(* IEC 61131-3 sources: std_i2980_v2.06_cp053/Source/IMM/ieccontrol/GlobalBaseArchives (part 9) *)

@END_Body

@@@BEG_Comment@@@
@TL(3)
This Algo receives the evCheckLocklist event,
checks the startconditions for the movement and outputs alarms if it is not allowed.
The movement itself is not started.
@@@END_Comment@@@

@BEG_Body
@TL(57)
(**************************************** WARNING ********************************************
 *** The KEBA Kemro K2 System including software is not intended for safety control tasks! ***
 ***                       For further information see Comment tab!                        ***
 *********************************************************************************************)

IF (evLockGroupEnableDisableData.DeviceIdReceiver.CompId = sv_DeviceId.CompId OR evLockGroupEnableDisableData.DeviceIdReceiver.CompId = cCompAll) AND
   (evLockGroupEnableDisableData.DeviceIdReceiver.IndexId = sv_DeviceId.IndexId OR evLockGroupEnableDisableData.DeviceIdReceiver.IndexId = cAllDevIndex) THEN

   //check all registered movements if the sent MoveDir and MoveId are equal
   FOR i := 1 TO sv_NumberOfMovements DO

      IF ((sv_Movements[i]^.MoveDir = evLockGroupEnableDisableData.MoveDir) OR (evLockGroupEnableDisableData.MoveDir = cMoveAll)) AND
         ((sv_Movements[i]^.MoveId = evLockGroupEnableDisableData.MoveId) OR (evLockGroupEnableDisableData.MoveId = cMoveAll)) THEN

         //check if this movement is a member of the sent lockgroup
         FOR j := 1 TO cMaxGroupLocks DO

            IF sv_Movements[i]^.LockGroups[j] = evLockGroupEnableDisableData.LockGroup THEN
               IF evLockGroupEnableDisableData.Mode = nLockGroupDisable THEN
                  mDisabledLockGroups[i][j] := TRUE;
               ELSE
                  mDisabledLockGroups[i][j] := FALSE;
               END_IF;

               IF sv_TraceLevel.bLockUnlock THEN
                  IF mDisabledLockGroups[i][j] THEN
                     sMode := ' disabled';
                  ELSE
                     sMode := ' enabled';
                  END_IF;

                  fbDebugTrace(CONCAT('lockgroup ', DINT_TO_STRING(evLockGroupEnableDisableData.LockGroup), ' of movement ',
                        DINT_TO_STRING(sv_Movements[i]^.MoveDir), '/', DINT_TO_STRING(sv_Movements[i]^.MoveId),
                        sMode, ' by Device ', DINT_TO_STRING(evLockGroupEnableDisableData.DeviceIdSender.CompId),
                        '.', DINT_TO_STRING(evLockGroupEnableDisableData.DeviceIdSender.IndexId)));
               END_IF;

               //update locklist
               abLockList.aUpdateLockDisable.Entry.DeviceIdSender := evLockGroupEnableDisableData.DeviceIdSender;
               abLockList.aUpdateLockDisable.Entry.MoveDir := sv_Movements[i]^.MoveDir;
               abLockList.aUpdateLockDisable.Entry.MoveId := sv_Movements[i]^.MoveId;
               abLockList.aUpdateLockDisable.Entry.Alarm := evLockGroupEnableDisableData.Alarm;
               abLockList.aUpdateLockDisable.bDisable := mDisabledLockGroups[i][j];
               abLockList.aUpdateLockDisable();
               EXIT;
            END_IF;

         END_FOR;  //end_for check lockgroups of the movement
      END_IF;  //end_if MoveDir and MoveId fit to event data
   END_FOR; //end_for check all movements

END_IF;

@END_Body

@@@BEG_Comment@@@
@TL(3)
receives evLockGroupEnableDisable event and updates locklist
if a registered movement of this function unit is a member of the
specified lockgroup
@@@END_Comment@@@
@END_Body

@END_Contents

(* ---- ABDeviceRegister.pu ---- *)
(*
@h    ! WARNING !
@h    The Kemro K2 system (including software) only meets category B according to EN 954-1,
@h    thus it is not intended for usage in safety-relevant control applications in the field
@h    of personal safety (e.g. emergency stop).
@h    To implement potentially necessary safety-relevant control tasks, always use additional
@h    external safety devices that are intended for the particular purpose, and meet the necessary
@h    functional safety.
@h    For further information see EN 954-1 (EN ISO 13849-1) and/or the K2-x00 user manual, chapter
@h    "CE conformity, directives and standards".

Increments the registration counter and calls the deviceregistation after the registrationdelay is up.
Every instance of ABDeviceRegister gets another delaytime - to give the other FUs time to increment
the registration counter.
*)

IMPORT_OVER_LISTFILE
 ABRegisterDelay
, FBDeviceRegister

END_IMPORT

ALGORITHM_BLOCK ABDeviceRegister #DUMMY_EDIT_BLOCK

SYSTEM_VAR
 sv_iDevicesToRegister : DINT;
END_VAR

SYSTEM_OBJECT
 Task10ms : TASK;
END_OBJECT

(*
Deviceregistration
*)

PROCESS_ALGORITHM paInit ON Task10ms AUTOSTART

VAR
 abRegisterDelay : ABRegisterDelay;
 fbDeviceRegister : FBDeviceRegister;
END_VAR

(* IecGraph-Code *)

(* init step *)
INITIAL_STEP DELAY:
aGetDelayTime (P);
END_STEP

ACTION aGetDelayTime: #BEGIN_EDIT_BLOCK
sv_iDevicesToRegister := sv_iDevicesToRegister + 1;
abRegisterDelay.aGet();

;#END_EDIT_BLOCK END_ACTION (*aGetDelayTime*)

(* steps *)
STEP DEVICE_REG:
Action2 (P);
END_STEP

ACTION Action2: #BEGIN_EDIT_BLOCK
fbDeviceRegister();
STOP_PROCESS_ALGORITHM();

;#END_EDIT_BLOCK END_ACTION (*Action2*)

(* transitions *)
TRANSITION Trans1 FROM DELAY TO DEVICE_REG :=  #BEGIN_EDIT_BLOCK
DELAY.T >= abRegisterDelay.aGet.Time
;#END_EDIT_BLOCK
END_TRANSITION

(* end IecGraph-Code *)
(* sfc-code *)
(* end sfc-code *)

END_ALGORITHM

END_ALGORITHM_BLOCK

#END_OF_IEC_PART

@Puma @IecEditor 6 10 @Pou 25
@@@BEG_Comment@@@
@h    ! WARNING !
@h    The Kemro K2 system (including software) only meets category B according to EN 954-1,
@h    thus it is not intended for usage in safety-relevant control applications in the field
@h    of personal safety (e.g. emergency stop).
@h    To implement potentially necessary safety-relevant control tasks, always use additional
@h    external safety devices that are intended for the particular purpose, and meet the necessary
@h    functional safety.
@h    For further information see EN 954-1 (EN ISO 13849-1) and/or the K2-x00 user manual, chapter
@h    "CE conformity, directives and standards".

Increments the registration counter and calls the deviceregistation after the registrationdelay is up.
Every instance of ABDeviceRegister gets another delaytime - to give the other FUs time to increment
the registration counter.
@@@END_Comment@@@

@BEG_Contents

@BEG_Func
@RT(17)FuncTreeContainer
0
@END_Func

@BEG_Const
@RT(18)ConstTreeContainer
0
@END_Const

@BEG_Export

@BEG_Kind
@ALGORITHM_BLOCK @RT(16)ABDeviceRegister @STRUCTURED_TEXT
@RT(0) @RT(0) @RT(0)
@END_Kind

@BEG_Dcl
@RT(16)DclTreeContainer
2
@Var @RT(21)sv_iDevicesToRegister @RT(0) @T @F @DT @RT(4)DINT @RT(0) @T @T @BASIC 0 @F
@F @F
@T
@BEG_Attrib
3 @RT(0) @RT(0) @RT(0)
@END_Attrib
1 8 @F @F @F @F

@Var @RT(8)Task10ms @RT(0) @T @T @RENAMED 0 @T @T @DT @RT(4)TASK @RT(0) @T @T @BASIC 0 @F
@F @F
@T
@BEG_Attrib
3 @RT(0) @RT(0) @RT(0)
@END_Attrib
1 7 @F @F @F @F

@END_Dcl

@END_Export

@BEG_Body

1

@BEG_Export

@BEG_Algo
@PROCESS_ALGORITHM @RT(6)paInit @SEQUENTIAL_FLOW_CHART
@RT(0) @RT(0) @RT(8)Task10ms @T @F
@END_Algo

@BEG_Dcl
@RT(16)DclTreeContainer
2
@Var @RT(15)abRegisterDelay @RT(0) @T @T @DERIVED 0 @T @T @DT @RT(15)ABRegisterDelay @RT(0) @T @T @UNKNOWN 0 @F
@F @F
@T
@BEG_Attrib
3 @RT(0) @RT(0) @RT(0)
@END_Attrib
1 0 @F @F @F @F

@Var @RT(16)fbDeviceRegister @RT(0) @T @T @DERIVED 0 @T @T @DT @RT(16)FBDeviceRegister @RT(0) @T @T @UNKNOWN 0 @F
@F @F
@T
@BEG_Attrib
3 @RT(0) @RT(0) @RT(0)
@END_Attrib
1 0 @F @F @F @F

@END_Dcl

@END_Export

@BEG_SfcBody
5 5 4

@BEG_SfcData 2
@StepSeq @RT(4)sseq @F 3
@Step @RT(5)DELAY @F @T @F @F @RT(0) @F
@AcbCont @RT(7)unnamed @F 1
@Acb @RT(13)aGetDelayTime @F @T @RT(1)P @RT(0) @F @F @T @TL(3)
sv_iDevicesToRegister := sv_iDevicesToRegister + 1;
abRegisterDelay.aGet();

@F

@Trans @RT(6)Trans1 @F @T @F @F @T @T @TL(2)
DELAY.T >= abRegisterDelay.aGet.Time

@RT(6)Trans1 @F
@Step @RT(10)DEVICE_REG @F @F @F @F @RT(0) @F
@AcbCont @RT(7)unnamed @F 1
@Acb @RT(7)Action2 @F @T @RT(1)P @RT(0) @F @F @T @TL(3)
fbDeviceRegister();
STOP_PROCESS_ALGORITHM();

@F

@END_SfcData
@SaActions 0
@SaTrans 0
@SaExits 0
@END_SfcBody

@@@BEG_Comment@@@
@TL(1)
Deviceregistration
@@@END_Comment@@@
@END_Body

@END_Contents

(* ---- ABEndPosMon.pu ---- *)
(*
@h    ! WARNING !
@h    The Kemro K2 system (including software) only meets category B according to EN 954-1,
@h    thus it is not intended for usage in safety-relevant control applications in the field
@h    of personal safety (e.g. emergency stop).
@h    To implement potentially necessary safety-relevant control tasks, always use additional
@h    external safety devices that are intended for the particular purpose, and meet the necessary
@h    functional safety.
@h    For further information see EN 954-1 (EN ISO 13849-1) and/or the K2-x00 user manual, chapter
@h    "CE conformity, directives and standards".

This AB is used for endposition supervision.
There are two possibilities to detect if an endpoint is reached.
- a limit switch for the endposition is available
- the last point of the entered movement profile is reached
The AB can handle a standard movement profile and plast profile.

The AB gives the following results in this cases:
1) only a limit switch and no movement profile
   => endposition is reached if limit switch is true

2) movement profile and no limit switch
   => endposition is reached if actual position is lower or equal / bigger or equal
      (depending on the movedirection) than last last position of the profile;
      a given tolerance will also be considered

3) movement profile and limit switch available
   => endposition is reached if both criterias from above are fullfilled
*)

IMPORT_OVER_LISTFILE
 CHECK_REF
, tsEndPosData
, KAPPL_VisProfile
, KAPPL_VisProfilePlast

END_IMPORT

ALGORITHM_BLOCK ABEndPosMon #DUMMY_EDIT_BLOCK

SYSTEM_VAR
 sv_EndPosData : tsEndPosData;
 sv_bInitStart : BOOL;
END_VAR

SYSTEM_OBJECT
 TaskAnalog : TASK;
 PU_Task_7 : TASK;
END_OBJECT

VAR
 mpProfile : REFTO KAPPL_VisProfile;
 mpPlastProfile : REFTO KAPPL_VisProfilePlast;
 mpTolerance : REFTO REAL;
 mbReparam : BOOL;
END_VAR

(*
This block checks if the actual position is within a tolerance at the target position.
If this condition is met, "Position Reached" is signaled.
*)

PROCESS_ALGORITHM paRun ON TaskAnalog(3000)

VAR
 bTargetPosReached : BOOL;
 rTargetPos : REAL;
 bDirection : BOOL;
 rTriggerPos : REAL;
 pbDI : REFTO BOOL;
 bDIConnected : BOOL;
 bValidMoveProfile : BOOL;
 bValidPlastProfile : BOOL;
 bValidProfile : BOOL;
 bInvertDI : BOOL;
END_VAR
#BEGIN_EDIT_BLOCK
(**************************************** WARNING ********************************************
 *** The KEBA Kemro K2 System including software is not intended for safety control tasks! ***
 ***                       For further information see Comment tab!                        ***
 *********************************************************************************************)

IF mbReparam THEN

   mpProfile := sv_EndPosData.pProfile;
   bValidMoveProfile := CHECK_REF(mpProfile^);
   mpPlastProfile := sv_EndPosData.pPlastProfile;
   bValidPlastProfile := CHECK_REF(mpPlastProfile^);
   bValidProfile := bValidMoveProfile OR bValidPlastProfile;

   pbDI := sv_EndPosData.pbDI;
   bDIConnected := CHECK_REF(pbDI^);
   bInvertDI := sv_EndPosData.bInvertDI;

   //get target position and direction
   IF bValidMoveProfile THEN
      rTargetPos := MAX(0.0, mpProfile^.Profile.Points[(mpProfile^.Profile.iNoOfPoints+1)].rStartPos);
      bDirection := mpProfile^.Profile.Points[mpProfile^.Profile.iNoOfPoints+1].rStartPos > mpProfile^.Profile.Points[1].rStartPos;
   ELSIF bValidPlastProfile THEN
      rTargetPos := MAX(0.0, mpPlastProfile^.Profile.Points[(mpPlastProfile^.Profile.iNoOfPoints+1)].rStartPos);
      bDirection := TRUE;
   END_IF;

   IF bValidProfile THEN
      IF bDirection THEN
         rTriggerPos := rTargetPos - sv_EndPosData.rTolerance^;
      ELSE
         rTriggerPos := rTargetPos + sv_EndPosData.rTolerance^;
      END_IF;
   END_IF;

   mbReparam := FALSE;
END_IF;

//cyclic part
IF bValidProfile THEN
   IF bDirection THEN
      bTargetPosReached := (sv_EndPosData.rActPos^ > rTriggerPos);
   ELSE
      bTargetPosReached := (sv_EndPosData.rActPos^ < rTriggerPos);
   END_IF;
END_IF;

IF bValidProfile AND bDIConnected THEN
   // profile and DI connected
   sv_EndPosData.pbPosReached^ := bTargetPosReached AND (pbDI^ XOR bInvertDI);
ELSIF bValidProfile THEN
   //only profile connected
   sv_EndPosData.pbPosReached^ := bTargetPosReached;
ELSIF bDIConnected THEN
   //only DI connected
   sv_EndPosData.pbPosReached^ := pbDI^ XOR bInvertDI;
END_IF;

;#END_EDIT_BLOCK END_ALGORITHM

POSTUPDATE_ALGORITHM pParameterChanged ON PU_Task_7 WITH mpTolerance^,mpProfile^.Profile,mpPlastProfile^.Profile,sv_EndPosData.pProfile,sv_EndPosData.pPlastProfile,sv_EndPosData.pbDI,sv_EndPosData.bInvertDI

#BEGIN_EDIT_BLOCK
(**************************************** WARNING ********************************************
 *** The KEBA Kemro K2 System including software is not intended for safety control tasks! ***
 ***                       For further information see Comment tab!                        ***
 *********************************************************************************************)

mbReparam := TRUE;

;#END_EDIT_BLOCK END_ALGORITHM

POSTUPDATE_ALGORITHM pInit ON PU_Task_7 WITH sv_bInitStart

#BEGIN_EDIT_BLOCK
(**************************************** WARNING ********************************************
 *** The KEBA Kemro K2 System including software is not intended for safety control tasks! ***
 ***                       For further information see Comment tab!                        ***
 *********************************************************************************************)

mpTolerance := sv_EndPosData.rTolerance;
mbReparam := TRUE;

START_PROCESS_ALGORITHM(paRun);

;#END_EDIT_BLOCK END_ALGORITHM

END_ALGORITHM_BLOCK

#END_OF_IEC_PART

@Puma @IecEditor 6 97 @Pou 25
@@@BEG_Comment@@@
@h    ! WARNING !
@h    The Kemro K2 system (including software) only meets category B according to EN 954-1,
@h    thus it is not intended for usage in safety-relevant control applications in the field
@h    of personal safety (e.g. emergency stop).
@h    To implement potentially necessary safety-relevant control tasks, always use additional
@h    external safety devices that are intended for the particular purpose, and meet the necessary
@h    functional safety.
@h    For further information see EN 954-1 (EN ISO 13849-1) and/or the K2-x00 user manual, chapter
@h    "CE conformity, directives and standards".

This AB is used for endposition supervision.
There are two possibilities to detect if an endpoint is reached.
- a limit switch for the endposition is available
- the last point of the entered movement profile is reached
The AB can handle a standard movement profile and plast profile.

The AB gives the following results in this cases:
1) only a limit switch and no movement profile
   => endposition is reached if limit switch is true

2) movement profile and no limit switch
   => endposition is reached if actual position is lower or equal / bigger or equal
      (depending on the movedirection) than last last position of the profile;
      a given tolerance will also be considered

3) movement profile and limit switch available
   => endposition is reached if both criterias from above are fullfilled
@@@END_Comment@@@

@BEG_Contents

@BEG_Func
@RT(17)FuncTreeContainer
1
@Var @RT(9)CHECK_REF @RT(0) @T @T @DERIVED 0 @F @RT(23)KEBA_STANDARD_PROCEDURE @F
@T
@BEG_Attrib
0 @RT(0) @RT(0)
@END_Attrib
1 1 @F @F @F @F

@END_Func

@BEG_Const
@RT(18)ConstTreeContainer
0
@END_Const

@BEG_Export

@BEG_Kind
@ALGORITHM_BLOCK @RT(11)ABEndPosMon @STRUCTURED_TEXT
@RT(0) @RT(0) @RT(0)
@END_Kind

@BEG_Dcl
@RT(16)DclTreeContainer
8
@Var @RT(13)sv_EndPosData @RT(0) @T @T @DERIVED 0 @T @T @DT @RT(12)tsEndPosData @RT(0) @T @T @UNKNOWN 0 @F
@F @F
@T
@BEG_Attrib
3 @RT(0) @RT(0) @RT(0)
@END_Attrib
1 8 @F @F @F @F

@Var @RT(10)TaskAnalog @RT(0) @T @T @RENAMED 0 @T @T @DT @RT(4)TASK @RT(0) @T @T @BASIC 0 @F
@F @F
@T
@BEG_Attrib
3 @RT(0) @RT(0) @RT(0)
@END_Attrib
1 7 @F @F @F @F

@Var @RT(9)PU_Task_7 @RT(0) @T @T @RENAMED 0 @T @T @DT @RT(4)TASK @RT(0) @T @T @BASIC 0 @F
@F @F
@T
@BEG_Attrib
3 @RT(0) @RT(0) @RT(0)
@END_Attrib
1 7 @F @F @F @F

@Var @RT(13)sv_bInitStart @RT(0) @T @F @DT @RT(4)BOOL @RT(0) @T @T @BASIC 0 @F
@F @F
@T
@BEG_Attrib
3 @RT(0) @RT(0) @RT(0)
@END_Attrib
1 8 @F @F @F @F

@Var @RT(9)mpProfile @RT(0) @T @T @REFTO 0 @F @DERIVED 0 @T @T @DT @RT(16)KAPPL_VisProfile @RT(0) @T @T @UNKNOWN 0 @F
@F @F
@T
@BEG_Attrib
3 @RT(0) @RT(0) @RT(0)
@END_Attrib
1 0 @F @F @F @F

@Var @RT(14)mpPlastProfile @RT(0) @T @T @REFTO 0 @F @DERIVED 0 @T @T @DT @RT(21)KAPPL_VisProfilePlast @RT(0) @T @T @UNKNOWN 0 @F
@F @F
@T
@BEG_Attrib
3 @RT(0) @RT(0) @RT(0)
@END_Attrib
1 0 @F @F @F @F

@Var @RT(11)mpTolerance @RT(0) @T @T @REFTO 0 @T @DT @RT(4)REAL @RT(0) @T @T @BASIC 0 @F
@F @F
@T
@BEG_Attrib
3 @RT(0) @RT(0) @RT(0)
@END_Attrib
1 0 @F @F @F @F

@Var @RT(9)mbReparam @RT(0) @T @F @DT @RT(4)BOOL @RT(0) @T @T @BASIC 0 @F
@F @F
@T
@BEG_Attrib
3 @RT(0) @RT(0) @RT(0)
@END_Attrib
1 0 @F @F @F @F

@END_Dcl

@END_Export

@BEG_Body

3

@BEG_Export

@BEG_Algo
@PROCESS_ALGORITHM @RT(5)paRun @STRUCTURED_TEXT
@RT(0) @RT(0) @RT(16)TaskAnalog(3000) @F @F
@END_Algo

@BEG_Dcl
@RT(16)DclTreeContainer
10
@Var @RT(17)bTargetPosReached @RT(0) @T @F @DT @RT(4)BOOL @RT(0) @T @T @BASIC 0 @F
@F @F
@T
@BEG_Attrib
3 @RT(0) @RT(0) @RT(0)
@END_Attrib
1 0 @F @F @F @F

@Var @RT(10)rTargetPos @RT(0) @T @F @DT @RT(4)REAL @RT(0) @T @T @BASIC 0 @F
@F @F
@T
@BEG_Attrib
3 @RT(0) @RT(0) @RT(0)
@END_Attrib
1 0 @F @F @F @F

@Var @RT(10)bDirection @RT(0) @T @F @DT @RT(4)BOOL @RT(0) @T @T @BASIC 0 @F
@F @F
@T
@BEG_Attrib
3 @RT(0) @RT(0) @RT(0)
@END_Attrib
1 0 @F @F @F @F

@Var @RT(11)rTriggerPos @RT(0) @T @F @DT @RT(4)REAL @RT(0) @T @T @BASIC 0 @F
@F @F
@T
@BEG_Attrib
3 @RT(0) @RT(0) @RT(0)
@END_Attrib
1 0 @F @F @F @F

@Var @RT(4)pbDI @RT(0) @T @T @REFTO 0 @T @DT @RT(4)BOOL @RT(0) @T @T @BASIC 0 @F
@F @F
@T
@BEG_Attrib
3 @RT(0) @RT(0) @RT(0)
@END_Attrib
1 0 @F @F @F @F

@Var @RT(12)bDIConnected @RT(0) @T @F @DT @RT(4)BOOL @RT(0) @T @T @BASIC 0 @F
@F @F
@T
@BEG_Attrib
3 @RT(0) @RT(0) @RT(0)
@END_Attrib
1 0 @F @F @F @F

@Var @RT(17)bValidMoveProfile @RT(0) @T @F @DT @RT(4)BOOL @RT(0) @T @T @BASIC 0 @F
@F @F
@T
@BEG_Attrib
3 @RT(0) @RT(0) @RT(0)
@END_Attrib
1 0 @F @F @F @F

@Var @RT(18)bValidPlastProfile @RT(0) @T @F @DT @RT(4)BOOL @RT(0) @T @T @BASIC 0 @F
@F @F
@T
@BEG_Attrib
3 @RT(0) @RT(0) @RT(0)
@END_Attrib
1 0 @F @F @F @F

@Var @RT(13)bValidProfile @RT(0) @T @F @DT @RT(4)BOOL @RT(0) @T @T @BASIC 0 @F
@F @F
@T
@BEG_Attrib
3 @RT(0) @RT(0) @RT(0)
@END_Attrib
1 0 @F @F @F @F

@Var @RT(9)bInvertDI @RT(0) @T @F @DT @RT(4)BOOL @RT(0) @T @T @BASIC 0 @F
@F @F
@T
@BEG_Attrib
3 @RT(0) @RT(0) @RT(0)
@END_Attrib
1 0 @F @F @F @F

@END_Dcl

@END_Export

@BEG_Export

@BEG_Algo
@POSTUPDATE_ALGORITHM @RT(17)pParameterChanged @STRUCTURED_TEXT
@RT(0) @RT(149)mpTolerance^,mpProfile^.Profile,mpPlastProfile^.Profile,sv_EndPosData.pProfile,sv_EndPosData.pPlastProfile,sv_EndPosData.pbDI,sv_EndPosData.bInvertDI @RT(9)PU_Task_7 @F @F
@END_Algo

@BEG_Dcl
@RT(16)DclTreeContainer
0
@END_Dcl

@END_Export

@BEG_Export

@BEG_Algo
@POSTUPDATE_ALGORITHM @RT(5)pInit @STRUCTURED_TEXT
@RT(0) @RT(13)sv_bInitStart @RT(9)PU_Task_7 @F @F
@END_Algo

@BEG_Dcl
@RT(16)DclTreeContainer
0
@END_Dcl

@END_Export

@BEG_Body
@TL(58)
(**************************************** WARNING ********************************************
 *** The KEBA Kemro K2 System including software is not intended for safety control tasks! ***
 ***                       For further information see Comment tab!                        ***
 *********************************************************************************************)

IF mbReparam THEN

   mpProfile := sv_EndPosData.pProfile;
   bValidMoveProfile := CHECK_REF(mpProfile^);
   mpPlastProfile := sv_EndPosData.pPlastProfile;
   bValidPlastProfile := CHECK_REF(mpPlastProfile^);
   bValidProfile := bValidMoveProfile OR bValidPlastProfile;

   pbDI := sv_EndPosData.pbDI;
   bDIConnected := CHECK_REF(pbDI^);
   bInvertDI := sv_EndPosData.bInvertDI;

   //get target position and direction
   IF bValidMoveProfile THEN
      rTargetPos := MAX(0.0, mpProfile^.Profile.Points[(mpProfile^.Profile.iNoOfPoints+1)].rStartPos);
      bDirection := mpProfile^.Profile.Points[mpProfile^.Profile.iNoOfPoints+1].rStartPos > mpProfile^.Profile.Points[1].rStartPos;
   ELSIF bValidPlastProfile THEN
      rTargetPos := MAX(0.0, mpPlastProfile^.Profile.Points[(mpPlastProfile^.Profile.iNoOfPoints+1)].rStartPos);
      bDirection := TRUE;
   END_IF;

   IF bValidProfile THEN
      IF bDirection THEN
         rTriggerPos := rTargetPos - sv_EndPosData.rTolerance^;
      ELSE
         rTriggerPos := rTargetPos + sv_EndPosData.rTolerance^;
      END_IF;
   END_IF;

   mbReparam := FALSE;
END_IF;

//cyclic part
IF bValidProfile THEN
   IF bDirection THEN
      bTargetPosReached := (sv_EndPosData.rActPos^ > rTriggerPos);
   ELSE
      bTargetPosReached := (sv_EndPosData.rActPos^ < rTriggerPos);
   END_IF;
END_IF;

IF bValidProfile AND bDIConnected THEN
   // profile and DI connected
   sv_EndPosData.pbPosReached^ := bTargetPosReached AND (pbDI^ XOR bInvertDI);
ELSIF bValidProfile THEN
   //only profile connected
   sv_EndPosData.pbPosReached^ := bTargetPosReached;
ELSIF bDIConnected THEN
   //only DI connected
   sv_EndPosData.pbPosReached^ := pbDI^ XOR bInvertDI;
END_IF;

@END_Body

@@@BEG_Comment@@@
@TL(2)
This block checks if the actual position is within a tolerance at the target position.
If this condition is met, "Position Reached" is signaled.
@@@END_Comment@@@

@BEG_Body
@TL(7)
(**************************************** WARNING ********************************************
 *** The KEBA Kemro K2 System including software is not intended for safety control tasks! ***
 ***                       For further information see Comment tab!                        ***
 *********************************************************************************************)

mbReparam := TRUE;

@END_Body

@@@BEG_Comment@@@
@TL(0)

@@@END_Comment@@@

@BEG_Body
@TL(10)
(**************************************** WARNING ********************************************
 *** The KEBA Kemro K2 System including software is not intended for safety control tasks! ***
 ***                       For further information see Comment tab!                        ***
 *********************************************************************************************)

mpTolerance := sv_EndPosData.rTolerance;
mbReparam := TRUE;

START_PROCESS_ALGORITHM(paRun);

@END_Body

@@@BEG_Comment@@@
@TL(0)

@@@END_Comment@@@
@END_Body

@END_Contents

(* ---- ABEnvelop.pu ---- *)
(*
/*-------------------------------------------------------------------------
 *                   (c) 2015 by KEBA AG
 *                            Linz/AUSTRIA
 *                         All rights reserved
 *--------------------------------------------------------------------------*/
Implementation of limitation of output with maximum speed,limit position and
maxramp to limit position.

Limitation can be done in both directions (increasing/decreasing position).
*)

IMPORT_OVER_LISTFILE
 KCTRL_YXGen_RampType_Sin
, cInvalidVelocityParams
, cCycleTimeError
, KCTRL_YXGen_RampType_Square
, KCTRL_Ret_OK
, cNoValidParams
, cCyclicCalculationError
, cInvalidMovementLimits
, KCTRL_YXGen_LightA
, KCTRL_YXGenParam
, KCTRL_YXGen_Accelerations

END_IMPORT

ALGORITHM_BLOCK ABEnvelop #DUMMY_EDIT_BLOCK

VAR
 mdCycleTime : TIME;
 mrMaxVelocity : REAL;
 mrMaxVelocityFwd : REAL;
 mrMaxVelocityBwd : REAL;
 mrMaxAcceleration : REAL;
 mrLimitPosition : REAL (* position where the limitation ends(after this 0 is allowed) *);
 mrMaxPosition : REAL (* position where the limitation ends(after this 0 is allowed) *);
 mrMinPosition : REAL (* position where the limitation ends(after this 0 is allowed) *);
 mrStartLimitingPosition : REAL (* position where the limitation starts(before this maximum velocity is allowed) *);
 mrStartLimitingPositionFwd : REAL (* position where the limitation forward starts(before this maximum velocity is allowed) *);
 mrStartLimitingPositionBwd : REAL (* position where the limitation backward starts(before this maximum velocity is allowed) *);
 mbLimitRisingPos : BOOL (* TRUE: limitation happens when position value increases FALSE: limitation happens when position value decreases *);
 mbParamOK : BOOL;
 mbParamDualOK : BOOL;
 abKCTRL_YXGen : KCTRL_YXGen_LightA;
 abKCTRL_YXGenFwd : KCTRL_YXGen_LightA;
 abKCTRL_YXGenBwd : KCTRL_YXGen_LightA;
END_VAR

ALGORITHM aPar

VAR_INPUT
 rMaxVelocity : REAL (* max. velocity anywhere *);
 rMaxAcceleration : REAL (* max. acceleration for ramp down at end *);
 rLimitPosition : REAL (* limit position. after this position 0 velocity is output, before this position the output ramps down *);
 bLimitRisingPos : BOOL (* TRUE: limitation happens when position value increases FALSE: limitation happens when position value decreases *);
 bRampTypeSquare : BOOL (* TRUE: use square ramps FALSE: use sin ramps *);
 dDeadTime : TIME (* dead time *);
 dCycleTime : TIME (* cycle time of the task calling aRun *);
END_VAR

VAR_OUTPUT
 bError : BOOL (* error during param *);
 iErrorInfo : DINT (* additional error info *);
END_VAR

VAR
 YXGenParam : KCTRL_YXGenParam := (Mode:=(RampType:=KCTRL_YXGen_RampType_Sin),ProfilePoints:=(uNoOfPoints:=2));
 YXGenAccelerations : KCTRL_YXGen_Accelerations;
END_VAR
#BEGIN_EDIT_BLOCK
(**************************************** WARNING ********************************************
 *** The KEBA Kemro K2 System including software is not intended for safety control tasks! ***
 ***                       For further information see Comment tab!                        ***
 *********************************************************************************************)
bError := FALSE;
iErrorInfo := 0;
mbParamOK := FALSE;

mdCycleTime := dCycleTime;
mrMaxVelocity := rMaxVelocity;
mrMaxAcceleration := rMaxAcceleration;
mrLimitPosition := rLimitPosition;
mbLimitRisingPos := bLimitRisingPos;

IF (mrMaxAcceleration <= 0.0) OR (mrMaxVelocity <= 0.0) THEN
    bError := TRUE;
    iErrorInfo := cInvalidVelocityParams;
    RETURN;
ELSIF (mdCycleTime <= T#0s) THEN
    bError := TRUE;
    iErrorInfo := cCycleTimeError;
    RETURN;
END_IF;

IF (mbLimitRisingPos) THEN
   mrStartLimitingPosition := mrLimitPosition - 0.5 * mrMaxVelocity * mrMaxVelocity / mrMaxAcceleration;
ELSE
   mrStartLimitingPosition := mrLimitPosition + 0.5 * mrMaxVelocity * mrMaxVelocity / mrMaxAcceleration;
END_IF;

IF bRampTypeSquare THEN
   YXGenParam.Mode.RampType := KCTRL_YXGen_RampType_Square;
ELSE
   YXGenParam.Mode.RampType := KCTRL_YXGen_RampType_Sin;
END_IF;
YXGenParam.ProfilePoints.Point[1].rX := mrStartLimitingPosition;
YXGenParam.ProfilePoints.Point[1].rY := mrMaxVelocity;
YXGenParam.ProfilePoints.Point[2].rX := mrLimitPosition;
YXGenParam.ProfilePoints.Point[2].rY := 0.0;

abKCTRL_YXGen.Par(dCycleTime := mdCycleTime,
                  Param := YXGenParam);
abKCTRL_YXGen.ParDeadTime(dDeadTime := dDeadTime);

YXGenAccelerations.rStart := mrMaxAcceleration;
YXGenAccelerations.rStop := mrMaxAcceleration;
YXGenAccelerations.rSoft := mrMaxAcceleration;
abKCTRL_YXGen.ParAccelerations(Accelerations := YXGenAccelerations);

abKCTRL_YXGen.Init(rX0 := mrStartLimitingPosition,
                   rY0 := mrMaxVelocity);

IF (abKCTRL_YXGen.Par.parStatus <> KCTRL_Ret_OK) OR
   (abKCTRL_YXGen.ParDeadTime.parStatus <> KCTRL_Ret_OK) OR
   (abKCTRL_YXGen.ParAccelerations.parStatus <> KCTRL_Ret_OK) OR
   (abKCTRL_YXGen.Init.initStatus <> KCTRL_Ret_OK) THEN
   bError := TRUE;
   iErrorInfo := cInvalidVelocityParams;
   RETURN;
END_IF;

// parametrization finished with valid parameters
mbParamOK := TRUE;

;#END_EDIT_BLOCK END_ALGORITHM

ALGORITHM aRun

VAR_INPUT
 bStart : BOOL R_EDGE (* start of movement *);
 bStop : BOOL (* stop movement *);
 rActPosition : REAL (* actual position *);
END_VAR

VAR_OUTPUT
 rLimitVelocity : REAL (* maximum output velocity *);
 bError : BOOL (* error during param *);
 iErrorInfo : DINT (* additional error info *);
END_VAR

VAR
 bInit : BOOL (* it is necessary to call abKCTRL_YXGen.Init *);
END_VAR
#BEGIN_EDIT_BLOCK
(**************************************** WARNING ********************************************
 *** The KEBA Kemro K2 System including software is not intended for safety control tasks! ***
 ***                       For further information see Comment tab!                        ***
 *********************************************************************************************)
IF NOT mbParamOK THEN
   // settings not initialized
   bError := TRUE;
   iErrorInfo := cNoValidParams;
   rLimitVelocity := 0.0;
   RETURN;
END_IF;

IF bStart THEN
   abKCTRL_YXGen.Init(rX0 := mrStartLimitingPosition,
                      rY0 := mrMaxVelocity);
   IF (abKCTRL_YXGen.Init.initStatus <> KCTRL_Ret_OK) THEN
      bError := TRUE;
      iErrorInfo := cInvalidVelocityParams;
      rLimitVelocity := 0.0;
      RETURN;
   END_IF;
END_IF;

IF ((mbLimitRisingPos AND (rActPosition < mrStartLimitingPosition)) OR
    ((NOT mbLimitRisingPos) AND (rActPosition > mrStartLimitingPosition))) AND
   (NOT bStop) THEN
   // We are before the start of the limitation -> allow full output
   // We do not need to ask the YX generator for this
   rLimitVelocity := mrMaxVelocity;
   bInit := TRUE;
ELSE
   // We are in the zone where limiting occurs
   IF (bInit) THEN
      abKCTRL_YXGen.Init(rX0 := mrStartLimitingPosition,
                         rY0 := mrMaxVelocity);
      IF (abKCTRL_YXGen.Init.initStatus <> KCTRL_Ret_OK) THEN
            bError := TRUE;
            iErrorInfo := cInvalidVelocityParams;
            rLimitVelocity := 0.0;
            RETURN;
      END_IF;
      bInit := FALSE;
   END_IF;

   abKCTRL_YXGen.Calculate(rX := rActPosition,
                           bSoftStop := bStop);
   IF (abKCTRL_YXGen.Calculate.calcStatus <> KCTRL_Ret_OK) THEN
      bError := TRUE;
      iErrorInfo := cCyclicCalculationError;
      rLimitVelocity := 0.0;
      RETURN;
   END_IF;
   rLimitVelocity := abKCTRL_YXGen.Calculate.rY;
END_IF;

bError := FALSE;
iErrorInfo := 0;

;#END_EDIT_BLOCK END_ALGORITHM

ALGORITHM aParDual

VAR_INPUT
 rMaxVelocityFwd : REAL (* max. velocity move increasing position, > 0.0 *);
 rMaxVelocityBwd : REAL (* max. velocity  move decreasing position, > 0.0 *);
 rMaxAcceleration : REAL (* max. acceleration for ramp down at end, > 0.0 *);
 rLimitMinPosition : REAL (* min. position limit, at lower position velocity output bwd is 0 *);
 rLimitMaxPosition : REAL (* max. position limit, at higher position velocity output fwd is 0 *);
 bRampTypeSquare : BOOL (* TRUE: use square ramps FALSE: use sin ramps *);
 dDeadTime : TIME (* dead time *);
 dCycleTime : TIME (* cycle time of the task calling aRun *);
END_VAR

VAR_OUTPUT
 bError : BOOL (* error during param *);
 iErrorInfo : DINT (* additional error info *);
END_VAR

VAR
 YXGenParamFwd : KCTRL_YXGenParam := (Mode:=(RampType:=KCTRL_YXGen_RampType_Sin),ProfilePoints:=(uNoOfPoints:=2));
 YXGenParamBwd : KCTRL_YXGenParam := (Mode:=(RampType:=KCTRL_YXGen_RampType_Sin),ProfilePoints:=(uNoOfPoints:=2));
 YXGenAccelerations : KCTRL_YXGen_Accelerations;
END_VAR
#BEGIN_EDIT_BLOCK
(**************************************** WARNING ********************************************
 *** The KEBA Kemro K2 System including software is not intended for safety control tasks! ***
 ***                       For further information see Comment tab!                        ***
 *********************************************************************************************)
bError := FALSE;
iErrorInfo := 0;
mbParamDualOK := FALSE;

mdCycleTime := dCycleTime;
mrMaxVelocityFwd := rMaxVelocityFwd;
mrMaxVelocityBwd := rMaxVelocityBwd;
mrMaxAcceleration := rMaxAcceleration;
mrMaxPosition := rLimitMaxPosition;
mrMinPosition := rLimitMinPosition;

IF (mrMaxAcceleration <= 0.0) OR
   (mrMaxVelocityFwd <= 0.0) OR
   (mrMaxVelocityBwd <= 0.0) THEN
    bError := TRUE;
    iErrorInfo := cInvalidVelocityParams;
    RETURN;
ELSIF (mdCycleTime <= T#0s) THEN
    bError := TRUE;
    iErrorInfo := cCycleTimeError;
    RETURN;
ELSIF (mrMaxPosition  < mrMinPosition) THEN
    bError := TRUE;
    iErrorInfo := cInvalidMovementLimits;
    RETURN;
END_IF;

mrStartLimitingPositionFwd := mrMaxPosition - 0.5 * mrMaxVelocityFwd * mrMaxVelocityFwd / mrMaxAcceleration;
mrStartLimitingPositionBwd := mrMinPosition + 0.5 * mrMaxVelocityBwd * mrMaxVelocityBwd / mrMaxAcceleration;

IF bRampTypeSquare THEN
   YXGenParamFwd.Mode.RampType := KCTRL_YXGen_RampType_Square;
   YXGenParamBwd.Mode.RampType := KCTRL_YXGen_RampType_Square;
ELSE
   YXGenParamFwd.Mode.RampType := KCTRL_YXGen_RampType_Sin;
   YXGenParamBwd.Mode.RampType := KCTRL_YXGen_RampType_Sin;
END_IF;
YXGenParamFwd.ProfilePoints.Point[1].rX := mrStartLimitingPositionFwd;
YXGenParamFwd.ProfilePoints.Point[1].rY := mrMaxVelocityFwd;
YXGenParamFwd.ProfilePoints.Point[2].rX := mrMaxPosition;
YXGenParamFwd.ProfilePoints.Point[2].rY := 0.0;

YXGenParamBwd.ProfilePoints.Point[1].rX := mrStartLimitingPositionBwd;
YXGenParamBwd.ProfilePoints.Point[1].rY := mrMaxVelocityBwd;
YXGenParamBwd.ProfilePoints.Point[2].rX := mrMinPosition;
YXGenParamBwd.ProfilePoints.Point[2].rY := 0.0;

abKCTRL_YXGenFwd.Par(dCycleTime := mdCycleTime,
                     Param := YXGenParamFwd);
abKCTRL_YXGenFwd.ParDeadTime(dDeadTime := dDeadTime);

abKCTRL_YXGenBwd.Par(dCycleTime := mdCycleTime,
                     Param := YXGenParamBwd);
abKCTRL_YXGenBwd.ParDeadTime(dDeadTime := dDeadTime);

YXGenAccelerations.rStart := 1.0e6;
YXGenAccelerations.rStop := mrMaxAcceleration;
YXGenAccelerations.rSoft := mrMaxAcceleration;
abKCTRL_YXGenFwd.ParAccelerations(Accelerations := YXGenAccelerations);
abKCTRL_YXGenBwd.ParAccelerations(Accelerations := YXGenAccelerations);

abKCTRL_YXGenFwd.Init(rX0 := mrStartLimitingPositionFwd,
                      rY0 := mrMaxVelocityFwd);
abKCTRL_YXGenBwd.Init(rX0 := mrStartLimitingPositionBwd,
                      rY0 := mrMaxVelocityBwd);
IF (abKCTRL_YXGenFwd.Par.parStatus <> KCTRL_Ret_OK) OR
   (abKCTRL_YXGenFwd.ParDeadTime.parStatus <> KCTRL_Ret_OK) OR
   (abKCTRL_YXGenFwd.ParAccelerations.parStatus <> KCTRL_Ret_OK) OR
   (abKCTRL_YXGenFwd.Init.initStatus <> KCTRL_Ret_OK) OR
   (abKCTRL_YXGenBwd.Par.parStatus <> KCTRL_Ret_OK) OR
   (abKCTRL_YXGenBwd.ParDeadTime.parStatus <> KCTRL_Ret_OK) OR
   (abKCTRL_YXGenBwd.ParAccelerations.parStatus <> KCTRL_Ret_OK) OR
   (abKCTRL_YXGenBwd.Init.initStatus <> KCTRL_Ret_OK) THEN
   bError := TRUE;
   iErrorInfo := cInvalidVelocityParams;
END_IF;

// parametrization finished with valid parameters
mbParamDualOK := TRUE;

;#END_EDIT_BLOCK END_ALGORITHM

ALGORITHM aRunDual

VAR_INPUT
 bStart : BOOL R_EDGE (* start of movement *);
 bStop : BOOL (* stop movement *);
 rActPosition : REAL (* actual position *);
END_VAR

VAR_OUTPUT
 rLimitVelocityFwd : REAL (* maximum output velocity increasing position, >= 0.0 *);
 rLimitVelocityBwd : REAL (* maximum output velocity decreasing position, >= 0.0 *);
 bError : BOOL (* error during param *);
 iErrorInfo : DINT (* additional error info *);
END_VAR

VAR
 bInitFwd : BOOL (* it is necessary to call abKCTRL_YXGen.Init *);
 bInitBwd : BOOL (* it is necessary to call abKCTRL_YXGen.Init *);
END_VAR
#BEGIN_EDIT_BLOCK
(**************************************** WARNING ********************************************
 *** The KEBA Kemro K2 System including software is not intended for safety control tasks! ***
 ***                       For further information see Comment tab!                        ***
 *********************************************************************************************)
IF NOT mbParamDualOK THEN
   // settings not initialized
   bError := TRUE;
   iErrorInfo := cNoValidParams;
   rLimitVelocityFwd := 0.0;
   rLimitVelocityBwd := 0.0;
   RETURN;
END_IF;

IF bStart THEN
   abKCTRL_YXGenFwd.Init(rX0 := mrStartLimitingPositionFwd,
                         rY0 := 0.0);
   abKCTRL_YXGenFwd.Calculate(rX := rActPosition);

   abKCTRL_YXGenBwd.Init(rX0 := mrStartLimitingPositionBwd,
                         rY0 := 0.0);
   abKCTRL_YXGenBwd.Calculate(rX := rActPosition);

   IF (abKCTRL_YXGenFwd.Init.initStatus <> KCTRL_Ret_OK) OR
      (abKCTRL_YXGenBwd.Init.initStatus <> KCTRL_Ret_OK) OR
      (abKCTRL_YXGenFwd.Calculate.calcStatus <> KCTRL_Ret_OK) OR
      (abKCTRL_YXGenBwd.Calculate.calcStatus <> KCTRL_Ret_OK) THEN
      bError := TRUE;
      iErrorInfo := cInvalidVelocityParams;
      rLimitVelocityFwd := 0.0;
      rLimitVelocityBwd := 0.0;
      RETURN;
   END_IF;
END_IF;

// calc fwd limit
IF (rActPosition < mrStartLimitingPositionFwd) AND (NOT bStop) THEN
   // we are before the start of the limitation -> allow full output
   // we do not need to ask the YX generator for this
   rLimitVelocityFwd := mrMaxVelocityFwd;
   bInitFwd := TRUE;
ELSE
   // We are in the zone where limiting occurs
   IF (bInitFwd) THEN
      abKCTRL_YXGenFwd.Init(rX0 := mrStartLimitingPositionFwd,
                            rY0 := mrMaxVelocityFwd);
      IF (abKCTRL_YXGenFwd.Init.initStatus <> KCTRL_Ret_OK) THEN
            bError := TRUE;
            iErrorInfo := cInvalidVelocityParams;
            rLimitVelocityFwd := 0.0;
            rLimitVelocityBwd := 0.0;
            RETURN;
      END_IF;
      bInitFwd := FALSE;
   END_IF;

   abKCTRL_YXGenFwd.Calculate(rX := rActPosition,
                              bSoftStop := bStop);
   IF (abKCTRL_YXGenFwd.Calculate.calcStatus <> KCTRL_Ret_OK) THEN
      bError := TRUE;
      iErrorInfo := cCyclicCalculationError;
      rLimitVelocityFwd := 0.0;
      rLimitVelocityBwd := 0.0;
      RETURN;
   END_IF;
   rLimitVelocityFwd := abKCTRL_YXGenFwd.Calculate.rY;
END_IF;

// calc bwd limit
IF (rActPosition > mrStartLimitingPositionBwd) AND (NOT bStop) THEN
   // we are before the start of the limitation -> allow full output
   // we do not need to ask the YX generator for this
   rLimitVelocityBwd := mrMaxVelocityBwd;
   bInitBwd := TRUE;
ELSE
   // We are in the zone where limiting occurs
   IF (bInitBwd) THEN
      abKCTRL_YXGenBwd.Init(rX0 := mrStartLimitingPositionBwd,
                         rY0 := mrMaxVelocityBwd);
      IF (abKCTRL_YXGenBwd.Init.initStatus <> KCTRL_Ret_OK) THEN
            bError := TRUE;
            iErrorInfo := cInvalidVelocityParams;
            rLimitVelocityFwd := 0.0;
            rLimitVelocityBwd := 0.0;
            RETURN;
      END_IF;
      bInitBwd := FALSE;
   END_IF;

   abKCTRL_YXGenBwd.Calculate(rX := rActPosition,
                              bSoftStop := bStop);
   IF (abKCTRL_YXGenBwd.Calculate.calcStatus <> KCTRL_Ret_OK) THEN
      bError := TRUE;
      iErrorInfo := cCyclicCalculationError;
      rLimitVelocityFwd := 0.0;
      rLimitVelocityBwd := 0.0;
      RETURN;
   END_IF;
   rLimitVelocityBwd := abKCTRL_YXGenBwd.Calculate.rY;
END_IF;

bError := FALSE;
iErrorInfo := 0;

;#END_EDIT_BLOCK END_ALGORITHM

END_ALGORITHM_BLOCK

#END_OF_IEC_PART

@Puma @IecEditor 6 144 @Pou 25
@@@BEG_Comment@@@
/*-------------------------------------------------------------------------
 *                   (c) 2015 by KEBA AG
 *                            Linz/AUSTRIA
 *                         All rights reserved
 *--------------------------------------------------------------------------*/
Implementation of limitation of output with maximum speed,limit position and
maxramp to limit position.

Limitation can be done in both directions (increasing/decreasing position).
@@@END_Comment@@@

@BEG_Contents

@BEG_Func
@RT(17)FuncTreeContainer
0
@END_Func

@BEG_Const
@RT(18)ConstTreeContainer
8
@Var @RT(24)KCTRL_YXGen_RampType_Sin @RT(0) @T @T @DERIVED 0 @F @RT(20)KCTRL_YXGen_RampType @F
@T
@BEG_Attrib
0 @RT(1)2 @RT(0)
@END_Attrib
1 1 @F @F @F @F

@Var @RT(22)cInvalidVelocityParams @RT(0) @T @F @DT @RT(0) @RT(0) @T @T @UNKNOWN 0 @F
@F @F
@T
@BEG_Attrib
0 @RT(0) @RT(0)
@END_Attrib
1 1 @F @F @F @F

@Var @RT(15)cCycleTimeError @RT(0) @T @F @DT @RT(0) @RT(0) @T @T @UNKNOWN 0 @F
@F @F
@T
@BEG_Attrib
0 @RT(0) @RT(0)
@END_Attrib
1 1 @F @F @F @F

@Var @RT(27)KCTRL_YXGen_RampType_Square @RT(0) @T @T @DERIVED 0 @F @RT(20)KCTRL_YXGen_RampType @F
@T
@BEG_Attrib
0 @RT(1)1 @RT(0)
@END_Attrib
1 1 @F @F @F @F

@Var @RT(12)KCTRL_Ret_OK @RT(0) @T @T @DERIVED 0 @F @RT(9)KCTRL_Ret @F
@T
@BEG_Attrib
0 @RT(1)0 @RT(0)
@END_Attrib
1 1 @F @F @F @F

@Var @RT(14)cNoValidParams @RT(0) @T @F @DT @RT(0) @RT(0) @T @T @UNKNOWN 0 @F
@F @F
@T
@BEG_Attrib
0 @RT(0) @RT(0)
@END_Attrib
1 1 @F @F @F @F

@Var @RT(23)cCyclicCalculationError @RT(0) @T @F @DT @RT(0) @RT(0) @T @T @UNKNOWN 0 @F
@F @F
@T
@BEG_Attrib
0 @RT(0) @RT(0)
@END_Attrib
1 1 @F @F @F @F

@Var @RT(22)cInvalidMovementLimits @RT(0) @T @F @DT @RT(0) @RT(0) @T @T @UNKNOWN 0 @F
@F @F
@T
@BEG_Attrib
0 @RT(0) @RT(0)
@END_Attrib
1 1 @F @F @F @F

@END_Const

@BEG_Export

@BEG_Kind
@ALGORITHM_BLOCK @RT(9)ABEnvelop @STRUCTURED_TEXT
@RT(0) @RT(0) @RT(0)
@END_Kind

@BEG_Dcl
@RT(16)DclTreeContainer
17
@Var @RT(11)mdCycleTime @RT(0) @T @F @DT @RT(4)TIME @RT(0) @T @T @BASIC 0 @F
@F @F
@T
@BEG_Attrib
3 @RT(0) @RT(0) @RT(0)
@END_Attrib
1 0 @F @F @F @F

@Var @RT(13)mrMaxVelocity @RT(0) @T @F @DT @RT(4)REAL @RT(0) @T @T @BASIC 0 @F
@F @F
@T
@BEG_Attrib
3 @RT(0) @RT(0) @RT(0)
@END_Attrib
1 0 @F @F @F @F

@Var @RT(16)mrMaxVelocityFwd @RT(0) @T @F @DT @RT(4)REAL @RT(0) @T @T @BASIC 0 @F
@F @F
@T
@BEG_Attrib
3 @RT(0) @RT(0) @RT(0)
@END_Attrib
1 0 @F @F @F @F

@Var @RT(16)mrMaxVelocityBwd @RT(0) @T @F @DT @RT(4)REAL @RT(0) @T @T @BASIC 0 @F
@F @F
@T
@BEG_Attrib
3 @RT(0) @RT(0) @RT(0)
@END_Attrib
1 0 @F @F @F @F

@Var @RT(17)mrMaxAcceleration @RT(0) @T @F @DT @RT(4)REAL @RT(0) @T @T @BASIC 0 @F
@F @F
@T
@BEG_Attrib
3 @RT(0) @RT(0) @RT(0)
@END_Attrib
1 0 @F @F @F @F

@Var @RT(15)mrLimitPosition @RT(0) @T @F @DT @RT(4)REAL @RT(0) @T @T @BASIC 0 @F
@F @F
@T
@BEG_Attrib
3 @RT(0) @RT(59)position where the limitation ends(after this 0 is allowed) @RT(0)
@END_Attrib
1 0 @F @F @F @F

@Var @RT(13)mrMaxPosition @RT(0) @T @F @DT @RT(4)REAL @RT(0) @T @T @BASIC 0 @F
@F @F
@T
@BEG_Attrib
3 @RT(0) @RT(59)position where the limitation ends(after this 0 is allowed) @RT(0)
@END_Attrib
1 0 @F @F @F @F

@Var @RT(13)mrMinPosition @RT(0) @T @F @DT @RT(4)REAL @RT(0) @T @T @BASIC 0 @F
@F @F
@T
@BEG_Attrib
3 @RT(0) @RT(59)position where the limitation ends(after this 0 is allowed) @RT(0)
@END_Attrib
1 0 @F @F @F @F

@Var @RT(23)mrStartLimitingPosition @RT(0) @T @F @DT @RT(4)REAL @RT(0) @T @T @BASIC 0 @F
@F @F
@T
@BEG_Attrib
3 @RT(0) @RT(77)position where the limitation starts(before this maximum velocity is allowed) @RT(0)
@END_Attrib
1 0 @F @F @F @F

@Var @RT(26)mrStartLimitingPositionFwd @RT(0) @T @F @DT @RT(4)REAL @RT(0) @T @T @BASIC 0 @F
@F @F
@T
@BEG_Attrib
3 @RT(0) @RT(85)position where the limitation forward starts(before this maximum velocity is allowed) @RT(0)
@END_Attrib
1 0 @F @F @F @F

@Var @RT(26)mrStartLimitingPositionBwd @RT(0) @T @F @DT @RT(4)REAL @RT(0) @T @T @BASIC 0 @F
@F @F
@T
@BEG_Attrib
3 @RT(0) @RT(86)position where the limitation backward starts(before this maximum velocity is allowed) @RT(0)
@END_Attrib
1 0 @F @F @F @F

@Var @RT(16)mbLimitRisingPos @RT(0) @T @F @DT @RT(4)BOOL @RT(0) @T @T @BASIC 0 @F
@F @F
@T
@BEG_Attrib
3 @RT(0) @RT(110)TRUE: limitation happens when position value increases FALSE: limitation happens when position value decreases @RT(0)
@END_Attrib
1 0 @F @F @F @F

@Var @RT(9)mbParamOK @RT(0) @T @F @DT @RT(4)BOOL @RT(0) @T @T @BASIC 0 @F
@F @F
@T
@BEG_Attrib
3 @RT(0) @RT(0) @RT(0)
@END_Attrib
1 0 @F @F @F @F

@Var @RT(13)mbParamDualOK @RT(0) @T @F @DT @RT(4)BOOL @RT(0) @T @T @BASIC 0 @F
@F @F
@T
@BEG_Attrib
3 @RT(0) @RT(0) @RT(0)
@END_Attrib
1 0 @F @F @F @F

@Var @RT(13)abKCTRL_YXGen @RT(0) @T @T @DERIVED 0 @T @T @DT @RT(18)KCTRL_YXGen_LightA @RT(0) @T @T @UNKNOWN 0 @F
@F @F
@T
@BEG_Attrib
3 @RT(0) @RT(0) @RT(0)
@END_Attrib
1 0 @F @F @F @F

@Var @RT(16)abKCTRL_YXGenFwd @RT(0) @T @T @DERIVED 0 @T @T @DT @RT(18)KCTRL_YXGen_LightA @RT(0) @T @T @UNKNOWN 0 @F
@F @F
@T
@BEG_Attrib
3 @RT(0) @RT(0) @RT(0)
@END_Attrib
1 0 @F @F @F @F

@Var @RT(16)abKCTRL_YXGenBwd @RT(0) @T @T @DERIVED 0 @T @T @DT @RT(18)KCTRL_YXGen_LightA @RT(0) @T @T @UNKNOWN 0 @F
@F @F
@T
@BEG_Attrib
3 @RT(0) @RT(0) @RT(0)
@END_Attrib
1 0 @F @F @F @F

@END_Dcl

@END_Export

@BEG_Body

4

@BEG_Export

@BEG_Algo
@ALGORITHM @RT(4)aPar @STRUCTURED_TEXT
@RT(0) @RT(0) @RT(0) @F @F
@END_Algo

@BEG_Dcl
@RT(16)DclTreeContainer
11
@Var @RT(12)rMaxVelocity @RT(0) @T @F @DT @RT(4)REAL @RT(0) @T @T @BASIC 0 @F
@F @F
@T
@BEG_Attrib
3 @RT(0) @RT(22)max. velocity anywhere @RT(0)
@END_Attrib
1 1 @F @F @F @F

@Var @RT(16)rMaxAcceleration @RT(0) @T @F @DT @RT(4)REAL @RT(0) @T @T @BASIC 0 @F
@F @F
@T
@BEG_Attrib
3 @RT(0) @RT(38)max. acceleration for ramp down at end @RT(0)
@END_Attrib
1 1 @F @F @F @F

@Var @RT(14)rLimitPosition @RT(0) @T @F @DT @RT(4)REAL @RT(0) @T @T @BASIC 0 @F
@F @F
@T
@BEG_Attrib
3 @RT(0) @RT(100)limit position. after this position 0 velocity is output, before this position the output ramps down @RT(0)
@END_Attrib
1 1 @F @F @F @F

@Var @RT(15)bLimitRisingPos @RT(0) @T @F @DT @RT(4)BOOL @RT(0) @T @T @BASIC 0 @F
@F @F
@T
@BEG_Attrib
3 @RT(0) @RT(110)TRUE: limitation happens when position value increases FALSE: limitation happens when position value decreases @RT(0)
@END_Attrib
1 1 @F @F @F @F

@Var @RT(15)bRampTypeSquare @RT(0) @T @F @DT @RT(4)BOOL @RT(0) @T @T @BASIC 0 @F
@F @F
@T
@BEG_Attrib
3 @RT(0) @RT(43)TRUE: use square ramps FALSE: use sin ramps @RT(0)
@END_Attrib
1 1 @F @F @F @F

@Var @RT(9)dDeadTime @RT(0) @T @F @DT @RT(4)TIME @RT(0) @T @T @BASIC 0 @F
@F @F
@T
@BEG_Attrib
3 @RT(0) @RT(9)dead time @RT(0)
@END_Attrib
1 1 @F @F @F @F

@Var @RT(10)dCycleTime @RT(0) @T @F @DT @RT(4)TIME @RT(0) @T @T @BASIC 0 @F
@F @F
@T
@BEG_Attrib
3 @RT(0) @RT(35)cycle time of the task calling aRun @RT(0)
@END_Attrib
1 1 @F @F @F @F

@Var @RT(6)bError @RT(0) @T @F @DT @RT(4)BOOL @RT(0) @T @T @BASIC 0 @F
@F @F
@T
@BEG_Attrib
3 @RT(0) @RT(18)error during param @RT(0)
@END_Attrib
1 3 @F @F @F @F

@Var @RT(10)iErrorInfo @RT(0) @T @F @DT @RT(4)DINT @RT(0) @T @T @BASIC 0 @F
@F @F
@T
@BEG_Attrib
3 @RT(0) @RT(21)additional error info @RT(0)
@END_Attrib
1 3 @F @F @F @F

@Var @RT(10)YXGenParam @RT(0) @T @T @DERIVED 0 @T @T @DT @RT(16)KCTRL_YXGenParam @RT(0) @T @T @UNKNOWN 0 @F
@F @F
@T
@BEG_Attrib
3 @RT(76)(Mode:=(RampType:=KCTRL_YXGen_RampType_Sin),ProfilePoints:=(uNoOfPoints:=2)) @RT(0) @RT(0)
@END_Attrib
1 0 @F @F @F @F

@Var @RT(18)YXGenAccelerations @RT(0) @T @T @DERIVED 0 @T @T @DT @RT(25)KCTRL_YXGen_Accelerations @RT(0) @T @T @UNKNOWN 0 @F
@F @F
@T
@BEG_Attrib
3 @RT(0) @RT(0) @RT(0)
@END_Attrib
1 0 @F @F @F @F

@END_Dcl

@END_Export

@BEG_Export

@BEG_Algo
@ALGORITHM @RT(4)aRun @STRUCTURED_TEXT
@RT(0) @RT(0) @RT(0) @F @F
@END_Algo

@BEG_Dcl
@RT(16)DclTreeContainer
7
@Var @RT(6)bStart @RT(0) @T @F @DT @RT(11)BOOL R_EDGE @RT(0) @T @T @BASIC 0 @F
@F @F
@T
@BEG_Attrib
3 @RT(0) @RT(17)start of movement @RT(0)
@END_Attrib
1 1 @F @F @F @F

@Var @RT(5)bStop @RT(0) @T @F @DT @RT(4)BOOL @RT(0) @T @T @BASIC 0 @F
@F @F
@T
@BEG_Attrib
3 @RT(0) @RT(13)stop movement @RT(0)
@END_Attrib
1 1 @F @F @F @F

@Var @RT(12)rActPosition @RT(0) @T @F @DT @RT(4)REAL @RT(0) @T @T @BASIC 0 @F
@F @F
@T
@BEG_Attrib
3 @RT(0) @RT(15)actual position @RT(0)
@END_Attrib
1 1 @F @F @F @F

@Var @RT(14)rLimitVelocity @RT(0) @T @F @DT @RT(4)REAL @RT(0) @T @T @BASIC 0 @F
@F @F
@T
@BEG_Attrib
3 @RT(0) @RT(23)maximum output velocity @RT(0)
@END_Attrib
1 3 @F @F @F @F

@Var @RT(6)bError @RT(0) @T @F @DT @RT(4)BOOL @RT(0) @T @T @BASIC 0 @F
@F @F
@T
@BEG_Attrib
3 @RT(0) @RT(18)error during param @RT(0)
@END_Attrib
1 3 @F @F @F @F

@Var @RT(10)iErrorInfo @RT(0) @T @F @DT @RT(4)DINT @RT(0) @T @T @BASIC 0 @F
@F @F
@T
@BEG_Attrib
3 @RT(0) @RT(21)additional error info @RT(0)
@END_Attrib
1 3 @F @F @F @F

@Var @RT(5)bInit @RT(0) @T @F @DT @RT(4)BOOL @RT(0) @T @T @BASIC 0 @F
@F @F
@T
@BEG_Attrib
3 @RT(0) @RT(42)it is necessary to call abKCTRL_YXGen.Init @RT(0)
@END_Attrib
1 0 @F @F @F @F

@END_Dcl

@END_Export

@BEG_Export

@BEG_Algo
@ALGORITHM @RT(8)aParDual @STRUCTURED_TEXT
@RT(0) @RT(0) @RT(0) @F @F
@END_Algo

@BEG_Dcl
@RT(16)DclTreeContainer
13
@Var @RT(15)rMaxVelocityFwd @RT(0) @T @F @DT @RT(4)REAL @RT(0) @T @T @BASIC 0 @F
@F @F
@T
@BEG_Attrib
3 @RT(0) @RT(45)max. velocity move increasing position, > 0.0 @RT(0)
@END_Attrib
1 1 @F @F @F @F

@Var @RT(15)rMaxVelocityBwd @RT(0) @T @F @DT @RT(4)REAL @RT(0) @T @T @BASIC 0 @F
@F @F
@T
@BEG_Attrib
3 @RT(0) @RT(46)max. velocity  move decreasing position, > 0.0 @RT(0)
@END_Attrib
1 1 @F @F @F @F

@Var @RT(16)rMaxAcceleration @RT(0) @T @F @DT @RT(4)REAL @RT(0) @T @T @BASIC 0 @F
@F @F
@T
@BEG_Attrib
3 @RT(0) @RT(45)max. acceleration for ramp down at end, > 0.0 @RT(0)
@END_Attrib
1 1 @F @F @F @F

@Var @RT(17)rLimitMinPosition @RT(0) @T @F @DT @RT(4)REAL @RT(0) @T @T @BASIC 0 @F
@F @F
@T
@BEG_Attrib
3 @RT(0) @RT(63)min. position limit, at lower position velocity output bwd is 0 @RT(0)
@END_Attrib
1 1 @F @F @F @F

@Var @RT(17)rLimitMaxPosition @RT(0) @T @F @DT @RT(4)REAL @RT(0) @T @T @BASIC 0 @F
@F @F
@T
@BEG_Attrib
3 @RT(0) @RT(64)max. position limit, at higher position velocity output fwd is 0 @RT(0)
@END_Attrib
1 1 @F @F @F @F

@Var @RT(15)bRampTypeSquare @RT(0) @T @F @DT @RT(4)BOOL @RT(0) @T @T @BASIC 0 @F
@F @F
@T
@BEG_Attrib
3 @RT(0) @RT(43)TRUE: use square ramps FALSE: use sin ramps @RT(0)
@END_Attrib
1 1 @F @F @F @F

@Var @RT(9)dDeadTime @RT(0) @T @F @DT @RT(4)TIME @RT(0) @T @T @BASIC 0 @F
@F @F
@T
@BEG_Attrib
3 @RT(0) @RT(9)dead time @RT(0)
@END_Attrib
1 1 @F @F @F @F

@Var @RT(10)dCycleTime @RT(0) @T @F @DT @RT(4)TIME @RT(0) @T @T @BASIC 0 @F
@F @F
@T
@BEG_Attrib
3 @RT(0) @RT(35)cycle time of the task calling aRun @RT(0)
@END_Attrib
1 1 @F @F @F @F

@Var @RT(6)bError @RT(0) @T @F @DT @RT(4)BOOL @RT(0) @T @T @BASIC 0 @F
@F @F
@T
@BEG_Attrib
3 @RT(0) @RT(18)error during param @RT(0)
@END_Attrib
1 3 @F @F @F @F

@Var @RT(10)iErrorInfo @RT(0) @T @F @DT @RT(4)DINT @RT(0) @T @T @BASIC 0 @F
@F @F
@T
@BEG_Attrib
3 @RT(0) @RT(21)additional error info @RT(0)
@END_Attrib
1 3 @F @F @F @F

@Var @RT(13)YXGenParamFwd @RT(0) @T @T @DERIVED 0 @T @T @DT @RT(16)KCTRL_YXGenParam @RT(0) @T @T @UNKNOWN 0 @F
@F @F
@T
@BEG_Attrib
3 @RT(76)(Mode:=(RampType:=KCTRL_YXGen_RampType_Sin),ProfilePoints:=(uNoOfPoints:=2)) @RT(0) @RT(0)
@END_Attrib
1 0 @F @F @F @F

@Var @RT(13)YXGenParamBwd @RT(0) @T @T @DERIVED 0 @T @T @DT @RT(16)KCTRL_YXGenParam @RT(0) @T @T @UNKNOWN 0 @F
@F @F
@T
@BEG_Attrib
3 @RT(76)(Mode:=(RampType:=KCTRL_YXGen_RampType_Sin),ProfilePoints:=(uNoOfPoints:=2)) @RT(0) @RT(0)
@END_Attrib
1 0 @F @F @F @F

@Var @RT(18)YXGenAccelerations @RT(0) @T @T @DERIVED 0 @T @T @DT @RT(25)KCTRL_YXGen_Accelerations @RT(0) @T @T @UNKNOWN 0 @F
@F @F
@T
@BEG_Attrib
3 @RT(0) @RT(0) @RT(0)
@END_Attrib
1 0 @F @F @F @F

@END_Dcl

@END_Export

@BEG_Export

@BEG_Algo
@ALGORITHM @RT(8)aRunDual @STRUCTURED_TEXT
@RT(0) @RT(0) @RT(0) @F @F
@END_Algo

@BEG_Dcl
@RT(16)DclTreeContainer
9
@Var @RT(6)bStart @RT(0) @T @F @DT @RT(11)BOOL R_EDGE @RT(0) @T @T @BASIC 0 @F
@F @F
@T
@BEG_Attrib
3 @RT(0) @RT(17)start of movement @RT(0)
@END_Attrib
1 1 @F @F @F @F

@Var @RT(5)bStop @RT(0) @T @F @DT @RT(4)BOOL @RT(0) @T @T @BASIC 0 @F
@F @F
@T
@BEG_Attrib
3 @RT(0) @RT(13)stop movement @RT(0)
@END_Attrib
1 1 @F @F @F @F

@Var @RT(12)rActPosition @RT(0) @T @F @DT @RT(4)REAL @RT(0) @T @T @BASIC 0 @F
@F @F
@T
@BEG_Attrib
3 @RT(0) @RT(15)actual position @RT(0)
@END_Attrib
1 1 @F @F @F @F

@Var @RT(17)rLimitVelocityFwd @RT(0) @T @F @DT @RT(4)REAL @RT(0) @T @T @BASIC 0 @F
@F @F
@T
@BEG_Attrib
3 @RT(0) @RT(51)maximum output velocity increasing position, >= 0.0 @RT(0)
@END_Attrib
1 3 @F @F @F @F

@Var @RT(17)rLimitVelocityBwd @RT(0) @T @F @DT @RT(4)REAL @RT(0) @T @T @BASIC 0 @F
@F @F
@T
@BEG_Attrib
3 @RT(0) @RT(51)maximum output velocity decreasing position, >= 0.0 @RT(0)
@END_Attrib
1 3 @F @F @F @F

@Var @RT(6)bError @RT(0) @T @F @DT @RT(4)BOOL @RT(0) @T @T @BASIC 0 @F
@F @F
@T
@BEG_Attrib
3 @RT(0) @RT(18)error during param @RT(0)
@END_Attrib
1 3 @F @F @F @F

@Var @RT(10)iErrorInfo @RT(0) @T @F @DT @RT(4)DINT @RT(0) @T @T @BASIC 0 @F
@F @F
@T
@BEG_Attrib
3 @RT(0) @RT(21)additional error info @RT(0)
@END_Attrib
1 3 @F @F @F @F

@Var @RT(8)bInitFwd @RT(0) @T @F @DT @RT(4)BOOL @RT(0) @T @T @BASIC 0 @F
@F @F
@T
@BEG_Attrib
3 @RT(0) @RT(42)it is necessary to call abKCTRL_YXGen.Init @RT(0)
@END_Attrib
1 0 @F @F @F @F

@Var @RT(8)bInitBwd @RT(0) @T @F @DT @RT(4)BOOL @RT(0) @T @T @BASIC 0 @F
@F @F
@T
@BEG_Attrib
3 @RT(0) @RT(42)it is necessary to call abKCTRL_YXGen.Init @RT(0)
@END_Attrib
1 0 @F @F @F @F

@END_Dcl

@END_Export

@BEG_Body
@TL(65)
(**************************************** WARNING ********************************************
 *** The KEBA Kemro K2 System including software is not intended for safety control tasks! ***
 ***                       For further information see Comment tab!                        ***
 *********************************************************************************************)
bError := FALSE;
iErrorInfo := 0;
mbParamOK := FALSE;

mdCycleTime := dCycleTime;
mrMaxVelocity := rMaxVelocity;
mrMaxAcceleration := rMaxAcceleration;
mrLimitPosition := rLimitPosition;
mbLimitRisingPos := bLimitRisingPos;

IF (mrMaxAcceleration <= 0.0) OR (mrMaxVelocity <= 0.0) THEN
    bError := TRUE;
    iErrorInfo := cInvalidVelocityParams;
    RETURN;
ELSIF (mdCycleTime <= T#0s) THEN
    bError := TRUE;
    iErrorInfo := cCycleTimeError;
    RETURN;
END_IF;

IF (mbLimitRisingPos) THEN
   mrStartLimitingPosition := mrLimitPosition - 0.5 * mrMaxVelocity * mrMaxVelocity / mrMaxAcceleration;
ELSE
   mrStartLimitingPosition := mrLimitPosition + 0.5 * mrMaxVelocity * mrMaxVelocity / mrMaxAcceleration;
END_IF;

IF bRampTypeSquare THEN
   YXGenParam.Mode.RampType := KCTRL_YXGen_RampType_Square;
ELSE
   YXGenParam.Mode.RampType := KCTRL_YXGen_RampType_Sin;
END_IF;
YXGenParam.ProfilePoints.Point[1].rX := mrStartLimitingPosition;
YXGenParam.ProfilePoints.Point[1].rY := mrMaxVelocity;
YXGenParam.ProfilePoints.Point[2].rX := mrLimitPosition;
YXGenParam.ProfilePoints.Point[2].rY := 0.0;

abKCTRL_YXGen.Par(dCycleTime := mdCycleTime,
                  Param := YXGenParam);
abKCTRL_YXGen.ParDeadTime(dDeadTime := dDeadTime);

YXGenAccelerations.rStart := mrMaxAcceleration;
YXGenAccelerations.rStop := mrMaxAcceleration;
YXGenAccelerations.rSoft := mrMaxAcceleration;
abKCTRL_YXGen.ParAccelerations(Accelerations := YXGenAccelerations);

abKCTRL_YXGen.Init(rX0 := mrStartLimitingPosition,
                   rY0 := mrMaxVelocity);

IF (abKCTRL_YXGen.Par.parStatus <> KCTRL_Ret_OK) OR
   (abKCTRL_YXGen.ParDeadTime.parStatus <> KCTRL_Ret_OK) OR
   (abKCTRL_YXGen.ParAccelerations.parStatus <> KCTRL_Ret_OK) OR
   (abKCTRL_YXGen.Init.initStatus <> KCTRL_Ret_OK) THEN
   bError := TRUE;
   iErrorInfo := cInvalidVelocityParams;
   RETURN;
END_IF;

// parametrization finished with valid parameters
mbParamOK := TRUE;

@END_Body

@@@BEG_Comment@@@
@TL(0)

@@@END_Comment@@@

@BEG_Body
@TL(58)
(**************************************** WARNING ********************************************
 *** The KEBA Kemro K2 System including software is not intended for safety control tasks! ***
 ***                       For further information see Comment tab!                        ***
 *********************************************************************************************)
IF NOT mbParamOK THEN
   // settings not initialized
   bError := TRUE;
   iErrorInfo := cNoValidParams;
   rLimitVelocity := 0.0;
   RETURN;
END_IF;

IF bStart THEN
   abKCTRL_YXGen.Init(rX0 := mrStartLimitingPosition,
                      rY0 := mrMaxVelocity);
   IF (abKCTRL_YXGen.Init.initStatus <> KCTRL_Ret_OK) THEN
      bError := TRUE;
      iErrorInfo := cInvalidVelocityParams;
      rLimitVelocity := 0.0;
      RETURN;
   END_IF;
END_IF;

IF ((mbLimitRisingPos AND (rActPosition < mrStartLimitingPosition)) OR
    ((NOT mbLimitRisingPos) AND (rActPosition > mrStartLimitingPosition))) AND
   (NOT bStop) THEN
   // We are before the start of the limitation -> allow full output
   // We do not need to ask the YX generator for this
   rLimitVelocity := mrMaxVelocity;
   bInit := TRUE;
ELSE
   // We are in the zone where limiting occurs
   IF (bInit) THEN
      abKCTRL_YXGen.Init(rX0 := mrStartLimitingPosition,
                         rY0 := mrMaxVelocity);
      IF (abKCTRL_YXGen.Init.initStatus <> KCTRL_Ret_OK) THEN
            bError := TRUE;
            iErrorInfo := cInvalidVelocityParams;
            rLimitVelocity := 0.0;
            RETURN;
      END_IF;
      bInit := FALSE;
   END_IF;

   abKCTRL_YXGen.Calculate(rX := rActPosition,
                           bSoftStop := bStop);
   IF (abKCTRL_YXGen.Calculate.calcStatus <> KCTRL_Ret_OK) THEN
      bError := TRUE;
      iErrorInfo := cCyclicCalculationError;
      rLimitVelocity := 0.0;
      RETURN;
   END_IF;
   rLimitVelocity := abKCTRL_YXGen.Calculate.rY;
END_IF;

bError := FALSE;
iErrorInfo := 0;

@END_Body

@@@BEG_Comment@@@
@TL(0)

@@@END_Comment@@@

@BEG_Body
@TL(86)
(**************************************** WARNING ********************************************
 *** The KEBA Kemro K2 System including software is not intended for safety control tasks! ***
 ***                       For further information see Comment tab!                        ***
 *********************************************************************************************)
bError := FALSE;
iErrorInfo := 0;
mbParamDualOK := FALSE;

mdCycleTime := dCycleTime;
mrMaxVelocityFwd := rMaxVelocityFwd;
mrMaxVelocityBwd := rMaxVelocityBwd;
mrMaxAcceleration := rMaxAcceleration;
mrMaxPosition := rLimitMaxPosition;
mrMinPosition := rLimitMinPosition;

IF (mrMaxAcceleration <= 0.0) OR
   (mrMaxVelocityFwd <= 0.0) OR
   (mrMaxVelocityBwd <= 0.0) THEN
    bError := TRUE;
    iErrorInfo := cInvalidVelocityParams;
    RETURN;
ELSIF (mdCycleTime <= T#0s) THEN
    bError := TRUE;
    iErrorInfo := cCycleTimeError;
    RETURN;
ELSIF (mrMaxPosition  < mrMinPosition) THEN
    bError := TRUE;
    iErrorInfo := cInvalidMovementLimits;
    RETURN;
END_IF;

mrStartLimitingPositionFwd := mrMaxPosition - 0.5 * mrMaxVelocityFwd * mrMaxVelocityFwd / mrMaxAcceleration;
mrStartLimitingPositionBwd := mrMinPosition + 0.5 * mrMaxVelocityBwd * mrMaxVelocityBwd / mrMaxAcceleration;

IF bRampTypeSquare THEN
   YXGenParamFwd.Mode.RampType := KCTRL_YXGen_RampType_Square;
   YXGenParamBwd.Mode.RampType := KCTRL_YXGen_RampType_Square;
ELSE
   YXGenParamFwd.Mode.RampType := KCTRL_YXGen_RampType_Sin;
   YXGenParamBwd.Mode.RampType := KCTRL_YXGen_RampType_Sin;
END_IF;
YXGenParamFwd.ProfilePoints.Point[1].rX := mrStartLimitingPositionFwd;
YXGenParamFwd.ProfilePoints.Point[1].rY := mrMaxVelocityFwd;
YXGenParamFwd.ProfilePoints.Point[2].rX := mrMaxPosition;
YXGenParamFwd.ProfilePoints.Point[2].rY := 0.0;

YXGenParamBwd.ProfilePoints.Point[1].rX := mrStartLimitingPositionBwd;
YXGenParamBwd.ProfilePoints.Point[1].rY := mrMaxVelocityBwd;
YXGenParamBwd.ProfilePoints.Point[2].rX := mrMinPosition;
YXGenParamBwd.ProfilePoints.Point[2].rY := 0.0;

abKCTRL_YXGenFwd.Par(dCycleTime := mdCycleTime,
                     Param := YXGenParamFwd);
abKCTRL_YXGenFwd.ParDeadTime(dDeadTime := dDeadTime);

abKCTRL_YXGenBwd.Par(dCycleTime := mdCycleTime,
                     Param := YXGenParamBwd);
abKCTRL_YXGenBwd.ParDeadTime(dDeadTime := dDeadTime);

YXGenAccelerations.rStart := 1.0e6;
YXGenAccelerations.rStop := mrMaxAcceleration;
YXGenAccelerations.rSoft := mrMaxAcceleration;
abKCTRL_YXGenFwd.ParAccelerations(Accelerations := YXGenAccelerations);
abKCTRL_YXGenBwd.ParAccelerations(Accelerations := YXGenAccelerations);

abKCTRL_YXGenFwd.Init(rX0 := mrStartLimitingPositionFwd,
                      rY0 := mrMaxVelocityFwd);
abKCTRL_YXGenBwd.Init(rX0 := mrStartLimitingPositionBwd,
                      rY0 := mrMaxVelocityBwd);
IF (abKCTRL_YXGenFwd.Par.parStatus <> KCTRL_Ret_OK) OR
   (abKCTRL_YXGenFwd.ParDeadTime.parStatus <> KCTRL_Ret_OK) OR
   (abKCTRL_YXGenFwd.ParAccelerations.parStatus <> KCTRL_Ret_OK) OR
   (abKCTRL_YXGenFwd.Init.initStatus <> KCTRL_Ret_OK) OR
   (abKCTRL_YXGenBwd.Par.parStatus <> KCTRL_Ret_OK) OR
   (abKCTRL_YXGenBwd.ParDeadTime.parStatus <> KCTRL_Ret_OK) OR
   (abKCTRL_YXGenBwd.ParAccelerations.parStatus <> KCTRL_Ret_OK) OR
   (abKCTRL_YXGenBwd.Init.initStatus <> KCTRL_Ret_OK) THEN
   bError := TRUE;
   iErrorInfo := cInvalidVelocityParams;
END_IF;

// parametrization finished with valid parameters
mbParamDualOK := TRUE;

@END_Body

@@@BEG_Comment@@@
@TL(0)

@@@END_Comment@@@

@BEG_Body
@TL(104)
(**************************************** WARNING ********************************************
 *** The KEBA Kemro K2 System including software is not intended for safety control tasks! ***
 ***                       For further information see Comment tab!                        ***
 *********************************************************************************************)
IF NOT mbParamDualOK THEN
   // settings not initialized
   bError := TRUE;
   iErrorInfo := cNoValidParams;
   rLimitVelocityFwd := 0.0;
   rLimitVelocityBwd := 0.0;
   RETURN;
END_IF;

IF bStart THEN
   abKCTRL_YXGenFwd.Init(rX0 := mrStartLimitingPositionFwd,
                         rY0 := 0.0);
   abKCTRL_YXGenFwd.Calculate(rX := rActPosition);

   abKCTRL_YXGenBwd.Init(rX0 := mrStartLimitingPositionBwd,
                         rY0 := 0.0);
   abKCTRL_YXGenBwd.Calculate(rX := rActPosition);

   IF (abKCTRL_YXGenFwd.Init.initStatus <> KCTRL_Ret_OK) OR
      (abKCTRL_YXGenBwd.Init.initStatus <> KCTRL_Ret_OK) OR
      (abKCTRL_YXGenFwd.Calculate.calcStatus <> KCTRL_Ret_OK) OR
      (abKCTRL_YXGenBwd.Calculate.calcStatus <> KCTRL_Ret_OK) THEN
      bError := TRUE;
      iErrorInfo := cInvalidVelocityParams;
      rLimitVelocityFwd := 0.0;
      rLimitVelocityBwd := 0.0;
      RETURN;
   END_IF;
END_IF;

// calc fwd limit
IF (rActPosition < mrStartLimitingPositionFwd) AND (NOT bStop) THEN
   // we are before the start of the limitation -> allow full output
   // we do not need to ask the YX generator for this
   rLimitVelocityFwd := mrMaxVelocityFwd;
   bInitFwd := TRUE;
ELSE
   // We are in the zone where limiting occurs
   IF (bInitFwd) THEN
      abKCTRL_YXGenFwd.Init(rX0 := mrStartLimitingPositionFwd,
                            rY0 := mrMaxVelocityFwd);
      IF (abKCTRL_YXGenFwd.Init.initStatus <> KCTRL_Ret_OK) THEN
            bError := TRUE;
            iErrorInfo := cInvalidVelocityParams;
            rLimitVelocityFwd := 0.0;
            rLimitVelocityBwd := 0.0;
            RETURN;
      END_IF;
      bInitFwd := FALSE;
   END_IF;

   abKCTRL_YXGenFwd.Calculate(rX := rActPosition,
                              bSoftStop := bStop);
   IF (abKCTRL_YXGenFwd.Calculate.calcStatus <> KCTRL_Ret_OK) THEN
      bError := TRUE;
      iErrorInfo := cCyclicCalculationError;
      rLimitVelocityFwd := 0.0;
      rLimitVelocityBwd := 0.0;
      RETURN;
   END_IF;
   rLimitVelocityFwd := abKCTRL_YXGenFwd.Calculate.rY;
END_IF;

// calc bwd limit
IF (rActPosition > mrStartLimitingPositionBwd) AND (NOT bStop) THEN
   // we are before the start of the limitation -> allow full output
   // we do not need to ask the YX generator for this
   rLimitVelocityBwd := mrMaxVelocityBwd;
   bInitBwd := TRUE;
ELSE
   // We are in the zone where limiting occurs
   IF (bInitBwd) THEN
      abKCTRL_YXGenBwd.Init(rX0 := mrStartLimitingPositionBwd,
                         rY0 := mrMaxVelocityBwd);
      IF (abKCTRL_YXGenBwd.Init.initStatus <> KCTRL_Ret_OK) THEN
            bError := TRUE;
            iErrorInfo := cInvalidVelocityParams;
            rLimitVelocityFwd := 0.0;
            rLimitVelocityBwd := 0.0;
            RETURN;
      END_IF;
      bInitBwd := FALSE;
   END_IF;

   abKCTRL_YXGenBwd.Calculate(rX := rActPosition,
                              bSoftStop := bStop);
   IF (abKCTRL_YXGenBwd.Calculate.calcStatus <> KCTRL_Ret_OK) THEN
      bError := TRUE;
      iErrorInfo := cCyclicCalculationError;
      rLimitVelocityFwd := 0.0;
      rLimitVelocityBwd := 0.0;
      RETURN;
   END_IF;
   rLimitVelocityBwd := abKCTRL_YXGenBwd.Calculate.rY;
END_IF;

bError := FALSE;
iErrorInfo := 0;

@END_Body

@@@BEG_Comment@@@
@TL(0)

@@@END_Comment@@@
@END_Body

@END_Contents

(* ---- ABHoldScrap.pu ---- *)
(*
@h    ! WARNING !
@h    The Kemro K2 system (including software) only meets category B according to EN 954-1,
@h    thus it is not intended for usage in safety-relevant control applications in the field
@h    of personal safety (e.g. emergency stop).
@h    To implement potentially necessary safety-relevant control tasks, always use additional
@h    external safety devices that are intended for the particular purpose, and meet the necessary
@h    functional safety.
@h    For further information see EN 954-1 (EN ISO 13849-1) and/or the K2-x00 user manual, chapter
@h    "CE conformity, directives and standards".

This AB handles evHoldScrap events.
If a evHoldScrap event is received, the device will be deactivated (set sv_bDeviceActivated to FALSE).
As a result this device will not be started during the rest of the autocycle.

After the operation has changed from HA or FA to manual, the device is activated again.
This reactivation is only done if the device was activated before the evHoldScrap event was received.
*)

IMPORT_OVER_LISTFILE
 tevHoldScrap
, tnOperationMode
, tevHoldScrapData

END_IMPORT

ALGORITHM_BLOCK ABHoldScrap #DUMMY_EDIT_BLOCK

SYSTEM_VAR
 sv_bDeviceActivated : BOOL;
 sv_OperationMode : tnOperationMode;
END_VAR

SYSTEM_OBJECT
 EV_Task_7 : TASK;
 evHoldScrap : tevHoldScrap;
 PU_Task_7 : TASK;
 TaskMid : TASK;
END_OBJECT

VAR
 miEventCount : DINT;
END_VAR

VAR RETAIN
 mbActivated : BOOL;
END_VAR

EVENT_ALGORITHM evaHoldScrap ON EV_Task_7 WITH evHoldScrap

VAR_INPUT
 evHoldScrapData : tevHoldScrapData;
END_VAR
#BEGIN_EDIT_BLOCK
(**************************************** WARNING ********************************************
 *** The KEBA Kemro K2 System including software is not intended for safety control tasks! ***
 ***                       For further information see Comment tab!                        ***
 *********************************************************************************************)

miEventCount := miEventCount + 1;
IF (miEventCount = 1) THEN
   //save status of activated flag when first "hold scrap" event is received
   mbActivated := sv_bDeviceActivated;
END_IF;

sv_bDeviceActivated := FALSE;

;#END_EDIT_BLOCK END_ALGORITHM

POSTUPDATE_ALGORITHM pOperationMode ON PU_Task_7 WITH sv_OperationMode

#BEGIN_EDIT_BLOCK
(**************************************** WARNING ********************************************
 *** The KEBA Kemro K2 System including software is not intended for safety control tasks! ***
 ***                       For further information see Comment tab!                        ***
 *********************************************************************************************)

IF (sv_OperationMode < nHalfAutomatic) THEN
   IF mbActivated THEN
      //device was activated before "hold scrap" was received
      //->reactivate the device
      sv_bDeviceActivated := TRUE;
   END_IF;

   //reset event counter
   miEventCount := 0;
END_IF;

;#END_EDIT_BLOCK END_ALGORITHM

PROCESS_ALGORITHM paInit ON TaskMid AUTOSTART

#BEGIN_EDIT_BLOCK
(**************************************** WARNING ********************************************
 *** The KEBA Kemro K2 System including software is not intended for safety control tasks! ***
 ***                       For further information see Comment tab!                        ***
 *********************************************************************************************)

//compare retain falg with sv_bDeviceActivated because
//possibly the controller was switched off before end of autocycle
IF mbActivated AND NOT sv_bDeviceActivated THEN
   sv_bDeviceActivated := TRUE;
END_IF;

STOP_PROCESS_ALGORITHM();

;#END_EDIT_BLOCK END_ALGORITHM

END_ALGORITHM_BLOCK

#END_OF_IEC_PART

@Puma @IecEditor 6 145 @Pou 25
@@@BEG_Comment@@@
@h    ! WARNING !
@h    The Kemro K2 system (including software) only meets category B according to EN 954-1,
@h    thus it is not intended for usage in safety-relevant control applications in the field
@h    of personal safety (e.g. emergency stop).
@h    To implement potentially necessary safety-relevant control tasks, always use additional
@h    external safety devices that are intended for the particular purpose, and meet the necessary
@h    functional safety.
@h    For further information see EN 954-1 (EN ISO 13849-1) and/or the K2-x00 user manual, chapter
@h    "CE conformity, directives and standards".

This AB handles evHoldScrap events.
If a evHoldScrap event is received, the device will be deactivated (set sv_bDeviceActivated to FALSE).
As a result this device will not be started during the rest of the autocycle.

After the operation has changed from HA or FA to manual, the device is activated again.
This reactivation is only done if the device was activated before the evHoldScrap event was received.
@@@END_Comment@@@

@BEG_Contents

@BEG_Func
@RT(17)FuncTreeContainer
0
@END_Func

@BEG_Const
@RT(18)ConstTreeContainer
0
@END_Const

@BEG_Export

@BEG_Kind
@ALGORITHM_BLOCK @RT(11)ABHoldScrap @STRUCTURED_TEXT
@RT(0) @RT(0) @RT(0)
@END_Kind

@BEG_Dcl
@RT(16)DclTreeContainer
8
@Var @RT(9)EV_Task_7 @RT(0) @T @T @RENAMED 0 @T @T @DT @RT(4)TASK @RT(0) @T @T @BASIC 0 @F
@F @F
@T
@BEG_Attrib
3 @RT(0) @RT(0) @RT(0)
@END_Attrib
1 7 @F @F @F @F

@Var @RT(11)evHoldScrap @RT(0) @T @T @RENAMED 0 @T @T @DT @RT(12)tevHoldScrap @RT(0) @T @T @UNKNOWN 0 @F
@F @F
@T
@BEG_Attrib
3 @RT(0) @RT(0) @RT(0)
@END_Attrib
1 7 @F @F @F @F

@Var @RT(19)sv_bDeviceActivated @RT(0) @T @F @DT @RT(4)BOOL @RT(0) @T @T @BASIC 0 @F
@F @F
@T
@BEG_Attrib
3 @RT(0) @RT(0) @RT(0)
@END_Attrib
1 8 @F @F @F @F

@Var @RT(9)PU_Task_7 @RT(0) @T @T @RENAMED 0 @T @T @DT @RT(4)TASK @RT(0) @T @T @BASIC 0 @F
@F @F
@T
@BEG_Attrib
3 @RT(0) @RT(0) @RT(0)
@END_Attrib
1 7 @F @F @F @F

@Var @RT(16)sv_OperationMode @RT(0) @T @T @RENAMED 0 @T @T @DT @RT(15)tnOperationMode @RT(0) @T @T @UNKNOWN 0 @F
@F @F
@T
@BEG_Attrib
3 @RT(0) @RT(0) @RT(0)
@END_Attrib
1 8 @F @F @F @F

@Var @RT(12)miEventCount @RT(0) @T @F @DT @RT(4)DINT @RT(0) @T @T @BASIC 0 @F
@F @F
@T
@BEG_Attrib
3 @RT(0) @RT(0) @RT(0)
@END_Attrib
1 0 @F @F @F @F

@Var @RT(11)mbActivated @RT(0) @T @F @DT @RT(4)BOOL @RT(0) @T @T @BASIC 0 @F
@F @F
@T
@BEG_Attrib
3 @RT(0) @RT(0) @RT(0)
@END_Attrib
1 11 @F @F @F @F

@Var @RT(7)TaskMid @RT(0) @T @T @RENAMED 0 @T @T @DT @RT(4)TASK @RT(0) @T @T @BASIC 0 @F
@F @F
@T
@BEG_Attrib
3 @RT(0) @RT(0) @RT(0)
@END_Attrib
1 7 @F @F @F @F

@END_Dcl

@END_Export

@BEG_Body

3

@BEG_Export

@BEG_Algo
@EVENT_ALGORITHM @RT(12)evaHoldScrap @STRUCTURED_TEXT
@RT(0) @RT(11)evHoldScrap @RT(9)EV_Task_7 @F @F
@END_Algo

@BEG_Dcl
@RT(16)DclTreeContainer
1
@Var @RT(15)evHoldScrapData @RT(0) @T @T @DERIVED 0 @F @RT(16)tevHoldScrapData @F
@T
@BEG_Attrib
3 @RT(0) @RT(0) @RT(0)
@END_Attrib
1 1 @F @F @F @F

@END_Dcl

@END_Export

@BEG_Export

@BEG_Algo
@POSTUPDATE_ALGORITHM @RT(14)pOperationMode @STRUCTURED_TEXT
@RT(0) @RT(16)sv_OperationMode @RT(9)PU_Task_7 @F @F
@END_Algo

@BEG_Dcl
@RT(16)DclTreeContainer
0
@END_Dcl

@END_Export

@BEG_Export

@BEG_Algo
@PROCESS_ALGORITHM @RT(6)paInit @STRUCTURED_TEXT
@RT(0) @RT(0) @RT(7)TaskMid @T @F
@END_Algo

@BEG_Dcl
@RT(16)DclTreeContainer
0
@END_Dcl

@END_Export

@BEG_Body
@TL(17)
(**************************************** WARNING ********************************************
 *** The KEBA Kemro K2 System including software is not intended for safety control tasks! ***
 ***                       For further information see Comment tab!                        ***
 *********************************************************************************************)

miEventCount := miEventCount + 1;
IF (miEventCount = 1) THEN
   //save status of activated flag when first "hold scrap" event is received
   mbActivated := sv_bDeviceActivated;
END_IF;

sv_bDeviceActivated := FALSE;

@END_Body

@@@BEG_Comment@@@
@TL(0)

@@@END_Comment@@@

@BEG_Body
@TL(17)
(**************************************** WARNING ********************************************
 *** The KEBA Kemro K2 System including software is not intended for safety control tasks! ***
 ***                       For further information see Comment tab!                        ***
 *********************************************************************************************)

IF (sv_OperationMode < nHalfAutomatic) THEN
   IF mbActivated THEN
      //device was activated before "hold scrap" was received
      //->reactivate the device
      sv_bDeviceActivated := TRUE;
   END_IF;

   //reset event counter
   miEventCount := 0;
END_IF;

@END_Body

@@@BEG_Comment@@@
@TL(0)

@@@END_Comment@@@

@BEG_Body
@TL(13)
(**************************************** WARNING ********************************************
 *** The KEBA Kemro K2 System including software is not intended for safety control tasks! ***
 ***                       For further information see Comment tab!                        ***
 *********************************************************************************************)

//compare retain falg with sv_bDeviceActivated because
//possibly the controller was switched off before end of autocycle
IF mbActivated AND NOT sv_bDeviceActivated THEN
   sv_bDeviceActivated := TRUE;
END_IF;

STOP_PROCESS_ALGORITHM();

@END_Body

@@@BEG_Comment@@@
@TL(0)

@@@END_Comment@@@
@END_Body

@END_Contents

(* ---- ABInterPosMon.pu ---- *)
IMPORT_OVER_LISTFILE
 tsInterPosData
, KCTRL_LimitSwitch
, KCTRL_LimitSwitch_Param

END_IMPORT

ALGORITHM_BLOCK ABInterPosMon #DUMMY_EDIT_BLOCK

SYSTEM_VAR
 sv_InterPosData : tsInterPosData;
 sv_bInitStart : BOOL;
END_VAR

SYSTEM_OBJECT
 TaskAnalog : TASK;
 TaskSlow : TASK;
 PU_Task_3 : TASK;
END_OBJECT

VAR
 abLimitSwitch : KCTRL_LimitSwitch;
 LimitSwitchParam : KCTRL_LimitSwitch_Param;
 mpTolerance : REFTO REAL;
 mprTargetPos : REFTO REAL;
END_VAR

PROCESS_ALGORITHM paRun ON TaskAnalog

#BEGIN_EDIT_BLOCK
(**************************************** WARNING ********************************************
 *** The KEBA Kemro K2 System including software is not intended for safety control tasks! ***
 ***                       For further information see Comment tab!                        ***
 *********************************************************************************************)

abLimitSwitch.Calculate(rX := sv_InterPosData.rActPos^);
sv_InterPosData.bPosReached^ := abLimitSwitch.Calculate.bY;

;#END_EDIT_BLOCK END_ALGORITHM

POSTUPDATE_ALGORITHM pParameterChanged ON PU_Task_3 WITH mpTolerance^,mprTargetPos^,sv_bInitStart

VAR
 bInitDone : BOOL;
END_VAR
#BEGIN_EDIT_BLOCK
(**************************************** WARNING ********************************************
 *** The KEBA Kemro K2 System including software is not intended for safety control tasks! ***
 ***                       For further information see Comment tab!                        ***
 *********************************************************************************************)

IF NOT bInitDone THEN
    mpTolerance := sv_InterPosData.rTolerance;
    mprTargetPos := sv_InterPosData.rTargetPos;
    bInitDone := TRUE;
END_IF;

LimitSwitchParam.rLimit := mprTargetPos^;
LimitSwitchParam.rDiffPEdge := sv_InterPosData.rTolerance^;
LimitSwitchParam.rDiffNEdge := sv_InterPosData.rTolerance^;

IF sv_InterPosData.bDirection THEN
    LimitSwitchParam.bModeInvert := FALSE;
ELSE
    LimitSwitchParam.bModeInvert := TRUE;
END_IF;

abLimitSwitch.Par(Param := LimitSwitchParam);
abLimitSwitch.Init(rX := sv_InterPosData.rActPos^);

abLimitSwitch.Calculate(rX := sv_InterPosData.rActPos^);
sv_InterPosData.bPosReached^ := abLimitSwitch.Calculate.bY;

START_PROCESS_ALGORITHM(paRun);

;#END_EDIT_BLOCK END_ALGORITHM

END_ALGORITHM_BLOCK

#END_OF_IEC_PART

@Puma @IecEditor 6 22 @Pou 25
@@@BEG_Comment@@@

@@@END_Comment@@@

@BEG_Contents

@BEG_Func
@RT(17)FuncTreeContainer
0
@END_Func

@BEG_Const
@RT(18)ConstTreeContainer
0
@END_Const

@BEG_Export

@BEG_Kind
@ALGORITHM_BLOCK @RT(13)ABInterPosMon @STRUCTURED_TEXT
@RT(0) @RT(0) @RT(0)
@END_Kind

@BEG_Dcl
@RT(16)DclTreeContainer
9
@Var @RT(15)sv_InterPosData @RT(0) @T @T @DERIVED 0 @T @T @DT @RT(14)tsInterPosData @RT(0) @T @T @UNKNOWN 0 @F
@F @F
@T
@BEG_Attrib
3 @RT(0) @RT(0) @RT(0)
@END_Attrib
1 8 @F @F @F @F

@Var @RT(10)TaskAnalog @RT(0) @T @T @RENAMED 0 @T @T @DT @RT(4)TASK @RT(0) @T @T @BASIC 0 @F
@F @F
@T
@BEG_Attrib
3 @RT(0) @RT(0) @RT(0)
@END_Attrib
1 7 @F @F @F @F

@Var @RT(8)TaskSlow @RT(0) @T @T @RENAMED 0 @T @T @DT @RT(4)TASK @RT(0) @T @T @BASIC 0 @F
@F @F
@T
@BEG_Attrib
3 @RT(0) @RT(0) @RT(0)
@END_Attrib
1 7 @F @F @F @F

@Var @RT(13)sv_bInitStart @RT(0) @T @F @DT @RT(4)BOOL @RT(0) @T @T @BASIC 0 @F
@F @F
@T
@BEG_Attrib
3 @RT(0) @RT(0) @RT(0)
@END_Attrib
1 8 @F @F @F @F

@Var @RT(13)abLimitSwitch @RT(0) @T @T @DERIVED 0 @T @T @DT @RT(17)KCTRL_LimitSwitch @RT(0) @T @T @UNKNOWN 0 @F
@F @F
@T
@BEG_Attrib
3 @RT(0) @RT(0) @RT(0)
@END_Attrib
1 0 @F @F @F @F

@Var @RT(16)LimitSwitchParam @RT(0) @T @T @DERIVED 0 @T @T @DT @RT(23)KCTRL_LimitSwitch_Param @RT(0) @T @T @UNKNOWN 0 @F
@F @F
@T
@BEG_Attrib
3 @RT(0) @RT(0) @RT(0)
@END_Attrib
1 0 @F @F @F @F

@Var @RT(11)mpTolerance @RT(0) @T @T @REFTO 0 @T @DT @RT(4)REAL @RT(0) @T @T @BASIC 0 @F
@F @F
@T
@BEG_Attrib
3 @RT(0) @RT(0) @RT(0)
@END_Attrib
1 0 @F @F @F @F

@Var @RT(12)mprTargetPos @RT(0) @T @T @REFTO 0 @T @DT @RT(4)REAL @RT(0) @T @T @BASIC 0 @F
@F @F
@T
@BEG_Attrib
3 @RT(0) @RT(0) @RT(0)
@END_Attrib
1 0 @F @F @F @F

@Var @RT(9)PU_Task_3 @RT(0) @T @T @RENAMED 0 @T @T @DT @RT(4)TASK @RT(0) @T @T @BASIC 0 @F
@F @F
@T
@BEG_Attrib
3 @RT(0) @RT(0) @RT(0)
@END_Attrib
1 7 @F @F @F @F

@END_Dcl

@END_Export

@BEG_Body

2

@BEG_Export

@BEG_Algo
@PROCESS_ALGORITHM @RT(5)paRun @STRUCTURED_TEXT
@RT(0) @RT(0) @RT(10)TaskAnalog @F @F
@END_Algo

@BEG_Dcl
@RT(16)DclTreeContainer
0
@END_Dcl

@END_Export

@BEG_Export

@BEG_Algo
@POSTUPDATE_ALGORITHM @RT(17)pParameterChanged @STRUCTURED_TEXT
@RT(0) @RT(40)mpTolerance^,mprTargetPos^,sv_bInitStart @RT(9)PU_Task_3 @F @F
@END_Algo

@BEG_Dcl
@RT(16)DclTreeContainer
1
@Var @RT(9)bInitDone @RT(0) @T @F @DT @RT(4)BOOL @RT(0) @T @T @BASIC 0 @F
@F @F
@T
@BEG_Attrib
3 @RT(0) @RT(0) @RT(0)
@END_Attrib
1 0 @F @F @F @F

@END_Dcl

@END_Export

@BEG_Body
@TL(10)
(**************************************** WARNING ********************************************
 *** The KEBA Kemro K2 System including software is not intended for safety control tasks! ***
 ***                       For further information see Comment tab!                        ***
 *********************************************************************************************)

abLimitSwitch.Calculate(rX := sv_InterPosData.rActPos^);
sv_InterPosData.bPosReached^ := abLimitSwitch.Calculate.bY;

@END_Body

@@@BEG_Comment@@@
@TL(0)

@@@END_Comment@@@

@BEG_Body
@TL(30)
(**************************************** WARNING ********************************************
 *** The KEBA Kemro K2 System including software is not intended for safety control tasks! ***
 ***                       For further information see Comment tab!                        ***
 *********************************************************************************************)

IF NOT bInitDone THEN
    mpTolerance := sv_InterPosData.rTolerance;
    mprTargetPos := sv_InterPosData.rTargetPos;
    bInitDone := TRUE;
END_IF;

LimitSwitchParam.rLimit := mprTargetPos^;
LimitSwitchParam.rDiffPEdge := sv_InterPosData.rTolerance^;
LimitSwitchParam.rDiffNEdge := sv_InterPosData.rTolerance^;

IF sv_InterPosData.bDirection THEN
    LimitSwitchParam.bModeInvert := FALSE;
ELSE
    LimitSwitchParam.bModeInvert := TRUE;
END_IF;

abLimitSwitch.Par(Param := LimitSwitchParam);
abLimitSwitch.Init(rX := sv_InterPosData.rActPos^);

abLimitSwitch.Calculate(rX := sv_InterPosData.rActPos^);
sv_InterPosData.bPosReached^ := abLimitSwitch.Calculate.bY;

START_PROCESS_ALGORITHM(paRun);

@END_Body

@@@BEG_Comment@@@
@TL(0)

@@@END_Comment@@@
@END_Body

@END_Contents

(* ---- ABLintabApply.pu ---- *)
(*
@h    ! WARNING !
@h    The Kemro K2 system (including software) only meets category B according to EN 954-1,
@h    thus it is not intended for usage in safety-relevant control applications in the field
@h    of personal safety (e.g. emergency stop).
@h    To implement potentially necessary safety-relevant control tasks, always use additional
@h    external safety devices that are intended for the particular purpose, and meet the necessary
@h    functional safety.
@h    For further information see EN 954-1 (EN ISO 13849-1) and/or the K2-x00 user manual, chapter
@h    "CE conformity, directives and standards".

apply a lintab to a output value
needed for converting absolute value outputs to percent / voltage
*)

IMPORT_OVER_LISTFILE
 KAPPL_LintabData
, KCTRL_Lintab_Light
, KCTRL_Lintab_Param_Light

END_IMPORT

ALGORITHM_BLOCK ABLintabApply #DUMMY_EDIT_BLOCK

SYSTEM_OBJECT
 EV_Task_1 : TASK;
END_OBJECT

VAR
 mpLintabPoints : REFTO KAPPL_LintabData;
 abKCTRL_Lintab : KCTRL_Lintab_Light;
 mParams : KCTRL_Lintab_Param_Light;
 mbReParam : BOOL (* lintab changed, need to reinitialize block on next aCalc/aCalcInv *);
 tmp : DINT;
END_VAR

ALGORITHM aInit

VAR_INPUT
 pLintab : REFTO KAPPL_LintabData;
 bLinearExtrapolation : BOOL;
END_VAR
#BEGIN_EDIT_BLOCK
(**************************************** WARNING ********************************************
 *** The KEBA Kemro K2 System including software is not intended for safety control tasks! ***
 ***                       For further information see Comment tab!                        ***
 *********************************************************************************************)

IF NOT CHECK_REF(pLintab^) THEN
   tmp := Print('ABLintabApply:aInit called with invalid Lintab');
   RETURN;
END_IF;
mpLintabPoints := pLintab;
mParams.LintabPoints := pLintab^.LintabPoints;
mParams.Mode.bLinearExtrapolation := bLinearExtrapolation;
mbReParam := TRUE;

;#END_EDIT_BLOCK END_ALGORITHM

POSTUPDATE_ALGORITHM pLintabchanged ON EV_Task_1(1) WITH mpLintabPoints^

#BEGIN_EDIT_BLOCK
(**************************************** WARNING ********************************************
 *** The KEBA Kemro K2 System including software is not intended for safety control tasks! ***
 ***                       For further information see Comment tab!                        ***
 *********************************************************************************************)

// remember for later that we need to reparam the lintab calculation block
mbReParam := TRUE;

;#END_EDIT_BLOCK END_ALGORITHM

(*
applies a lintab to the input value
*)

ALGORITHM aCalc

VAR_INPUT
 rX : REAL;
END_VAR

VAR_OUTPUT
 rY : REAL;
END_VAR
#BEGIN_EDIT_BLOCK
(**************************************** WARNING ********************************************
 *** The KEBA Kemro K2 System including software is not intended for safety control tasks! ***
 ***                       For further information see Comment tab!                        ***
 *********************************************************************************************)

IF mbReParam THEN
   mbReParam := FALSE;
   mParams.LintabPoints := mpLintabPoints^.LintabPoints;
   abKCTRL_Lintab.Par(Param := mParams);
   abKCTRL_Lintab.Init();
END_IF;

abKCTRL_Lintab.Calculate(rX := rX);
rY := abKCTRL_Lintab.Calculate.rY;

;#END_EDIT_BLOCK END_ALGORITHM

(*
applies a lintab to the input value
*)

ALGORITHM aCalcInv

VAR_OUTPUT
 rX : REAL;
END_VAR

VAR_INPUT
 rY : REAL;
END_VAR
#BEGIN_EDIT_BLOCK
(**************************************** WARNING ********************************************
 *** The KEBA Kemro K2 System including software is not intended for safety control tasks! ***
 ***                       For further information see Comment tab!                        ***
 *********************************************************************************************)

IF mbReParam THEN
   mbReParam := FALSE;
   mParams.LintabPoints := mpLintabPoints^.LintabPoints;
   abKCTRL_Lintab.Par(Param := mParams);
   abKCTRL_Lintab.Init();
END_IF;

abKCTRL_Lintab.CalculateInv(rY := rY);
rX := abKCTRL_Lintab.CalculateInv.rX;

;#END_EDIT_BLOCK END_ALGORITHM

END_ALGORITHM_BLOCK

#END_OF_IEC_PART

@Puma @IecEditor 6 30 @Pou 25
@@@BEG_Comment@@@
@h    ! WARNING !
@h    The Kemro K2 system (including software) only meets category B according to EN 954-1,
@h    thus it is not intended for usage in safety-relevant control applications in the field
@h    of personal safety (e.g. emergency stop).
@h    To implement potentially necessary safety-relevant control tasks, always use additional
@h    external safety devices that are intended for the particular purpose, and meet the necessary
@h    functional safety.
@h    For further information see EN 954-1 (EN ISO 13849-1) and/or the K2-x00 user manual, chapter
@h    "CE conformity, directives and standards".

apply a lintab to a output value
needed for converting absolute value outputs to percent / voltage
@@@END_Comment@@@

@BEG_Contents

@BEG_Func
@RT(17)FuncTreeContainer
0
@END_Func

@BEG_Const
@RT(18)ConstTreeContainer
0
@END_Const

@BEG_Export

@BEG_Kind
@ALGORITHM_BLOCK @RT(13)ABLintabApply @STRUCTURED_TEXT
@RT(0) @RT(0) @RT(0)
@END_Kind

@BEG_Dcl
@RT(16)DclTreeContainer
6
@Var @RT(14)mpLintabPoints @RT(0) @T @T @REFTO 0 @F @DERIVED 0 @T @T @DT @RT(16)KAPPL_LintabData @RT(0) @T @T @UNKNOWN 0 @F
@F @F
@T
@BEG_Attrib
3 @RT(0) @RT(0) @RT(0)
@END_Attrib
1 0 @F @F @F @F

@Var @RT(14)abKCTRL_Lintab @RT(0) @T @T @DERIVED 0 @T @T @DT @RT(18)KCTRL_Lintab_Light @RT(0) @T @T @UNKNOWN 0 @F
@F @F
@T
@BEG_Attrib
3 @RT(0) @RT(0) @RT(0)
@END_Attrib
1 0 @F @F @F @F

@Var @RT(7)mParams @RT(0) @T @T @DERIVED 0 @T @T @DT @RT(24)KCTRL_Lintab_Param_Light @RT(0) @T @T @UNKNOWN 0 @F
@F @F
@T
@BEG_Attrib
3 @RT(0) @RT(0) @RT(0)
@END_Attrib
1 0 @F @F @F @F

@Var @RT(9)mbReParam @RT(0) @T @T @RENAMED 0 @T @T @DT @RT(4)BOOL @RT(0) @T @T @BASIC 0 @F
@F @F
@T
@BEG_Attrib
3 @RT(0) @RT(65)lintab changed, need to reinitialize block on next aCalc/aCalcInv @RT(0)
@END_Attrib
1 0 @F @F @F @F

@Var @RT(3)tmp @RT(0) @T @F @DT @RT(4)DINT @RT(0) @T @T @BASIC 0 @F
@F @F
@T
@BEG_Attrib
3 @RT(0) @RT(0) @RT(0)
@END_Attrib
1 0 @F @F @F @F

@Var @RT(9)EV_Task_1 @RT(0) @T @T @RENAMED 0 @T @T @DT @RT(4)TASK @RT(0) @T @T @BASIC 0 @F
@F @F
@T
@BEG_Attrib
3 @RT(0) @RT(0) @RT(0)
@END_Attrib
1 7 @F @F @F @F

@END_Dcl

@END_Export

@BEG_Body

4

@BEG_Export

@BEG_Algo
@ALGORITHM @RT(5)aInit @STRUCTURED_TEXT
@RT(0) @RT(0) @RT(0) @F @F
@END_Algo

@BEG_Dcl
@RT(16)DclTreeContainer
2
@Var @RT(7)pLintab @RT(0) @T @T @REFTO 0 @F @DERIVED 0 @T @T @DT @RT(16)KAPPL_LintabData @RT(0) @T @T @UNKNOWN 0 @F
@F @F
@T
@BEG_Attrib
3 @RT(0) @RT(0) @RT(0)
@END_Attrib
1 1 @F @F @F @F

@Var @RT(20)bLinearExtrapolation @RT(0) @T @F @DT @RT(4)BOOL @RT(0) @T @T @BASIC 0 @F
@F @F
@T
@BEG_Attrib
3 @RT(0) @RT(0) @RT(0)
@END_Attrib
1 1 @F @F @F @F

@END_Dcl

@END_Export

@BEG_Export

@BEG_Algo
@POSTUPDATE_ALGORITHM @RT(14)pLintabchanged @STRUCTURED_TEXT
@RT(0) @RT(15)mpLintabPoints^ @RT(12)EV_Task_1(1) @F @F
@END_Algo

@BEG_Dcl
@RT(16)DclTreeContainer
0
@END_Dcl

@END_Export

@BEG_Export

@BEG_Algo
@ALGORITHM @RT(5)aCalc @STRUCTURED_TEXT
@RT(0) @RT(0) @RT(0) @F @F
@END_Algo

@BEG_Dcl
@RT(16)DclTreeContainer
2
@Var @RT(2)rX @RT(0) @T @F @DT @RT(4)REAL @RT(0) @T @T @BASIC 0 @F
@F @F
@T
@BEG_Attrib
3 @RT(0) @RT(0) @RT(0)
@END_Attrib
1 1 @F @F @F @F

@Var @RT(2)rY @RT(0) @T @F @DT @RT(4)REAL @RT(0) @T @T @BASIC 0 @F
@F @F
@T
@BEG_Attrib
3 @RT(0) @RT(0) @RT(0)
@END_Attrib
1 3 @F @F @F @F

@END_Dcl

@END_Export

@BEG_Export

@BEG_Algo
@ALGORITHM @RT(8)aCalcInv @STRUCTURED_TEXT
@RT(0) @RT(0) @RT(0) @F @F
@END_Algo

@BEG_Dcl
@RT(16)DclTreeContainer
2
@Var @RT(2)rX @RT(0) @T @F @DT @RT(4)REAL @RT(0) @T @T @BASIC 0 @F
@F @F
@T
@BEG_Attrib
3 @RT(0) @RT(0) @RT(0)
@END_Attrib
1 3 @F @F @F @F

@Var @RT(2)rY @RT(0) @T @F @DT @RT(4)REAL @RT(0) @T @T @BASIC 0 @F
@F @F
@T
@BEG_Attrib
3 @RT(0) @RT(0) @RT(0)
@END_Attrib
1 1 @F @F @F @F

@END_Dcl

@END_Export

@BEG_Body
@TL(14)
(**************************************** WARNING ********************************************
 *** The KEBA Kemro K2 System including software is not intended for safety control tasks! ***
 ***                       For further information see Comment tab!                        ***
 *********************************************************************************************)

IF NOT CHECK_REF(pLintab^) THEN
   tmp := Print('ABLintabApply:aInit called with invalid Lintab');
   RETURN;
END_IF;
mpLintabPoints := pLintab;
mParams.LintabPoints := pLintab^.LintabPoints;
mParams.Mode.bLinearExtrapolation := bLinearExtrapolation;
mbReParam := TRUE;

@END_Body

@@@BEG_Comment@@@
@TL(0)

@@@END_Comment@@@

@BEG_Body
@TL(8)
(**************************************** WARNING ********************************************
 *** The KEBA Kemro K2 System including software is not intended for safety control tasks! ***
 ***                       For further information see Comment tab!                        ***
 *********************************************************************************************)

// remember for later that we need to reparam the lintab calculation block
mbReParam := TRUE;

@END_Body

@@@BEG_Comment@@@
@TL(0)

@@@END_Comment@@@

@BEG_Body
@TL(16)
(**************************************** WARNING ********************************************
 *** The KEBA Kemro K2 System including software is not intended for safety control tasks! ***
 ***                       For further information see Comment tab!                        ***
 *********************************************************************************************)

IF mbReParam THEN
   mbReParam := FALSE;
   mParams.LintabPoints := mpLintabPoints^.LintabPoints;
   abKCTRL_Lintab.Par(Param := mParams);
   abKCTRL_Lintab.Init();
END_IF;

abKCTRL_Lintab.Calculate(rX := rX);
rY := abKCTRL_Lintab.Calculate.rY;

@END_Body

@@@BEG_Comment@@@
@TL(1)
applies a lintab to the input value
@@@END_Comment@@@

@BEG_Body
@TL(16)
(**************************************** WARNING ********************************************
 *** The KEBA Kemro K2 System including software is not intended for safety control tasks! ***
 ***                       For further information see Comment tab!                        ***
 *********************************************************************************************)

IF mbReParam THEN
   mbReParam := FALSE;
   mParams.LintabPoints := mpLintabPoints^.LintabPoints;
   abKCTRL_Lintab.Par(Param := mParams);
   abKCTRL_Lintab.Init();
END_IF;

abKCTRL_Lintab.CalculateInv(rY := rY);
rX := abKCTRL_Lintab.CalculateInv.rX;

@END_Body

@@@BEG_Comment@@@
@TL(1)
applies a lintab to the input value
@@@END_Comment@@@
@END_Body

@END_Contents
